LIN {X 0,Y 151.898,Z 448.046,A -85,B 0,C 180,E1 -25589.636,E2 -25589.636} C_VEL
LIN {X 0,Y 155.707,Z 455.378,A -85,B 0,C 180,E1 -25592.608,E2 -25592.608} C_VEL
LIN {X 0,Y 160.06,Z 464.974,A -85,B 0,C 180,E1 -25595.673,E2 -25595.673} C_VEL
LIN {X 0,Y 164.025,Z 475.268,A -85,B 0,C 180,E1 -25598.259,E2 -25598.259} C_VEL
LIN {X 0,Y 165.804,Z 480.611,A -85,B 0,C 180,E1 -25599.382,E2 -25599.382} C_VEL
LIN {X 0,Y 163.11,Z 515.862,A -85,B 0,C 180,E1 -25600.725,E2 -25600.725} C_VEL
LIN {X 0,Y 160.97,Z 529.245,A -85,B 0,C 180,E1 -25601.57,E2 -25601.57} C_VEL
LIN {X 0,Y 157.876,Z 541.895,A -85,B 0,C 180,E1 -25602.735,E2 -25602.735} C_VEL
LIN {X 0,Y 153.84,Z 554.553,A -85,B 0,C 180,E1 -25604.456,E2 -25604.456} C_VEL
LIN {X 0,Y 149.366,Z 565.815,A -85,B 0,C 180,E1 -25606.518,E2 -25606.518} C_VEL
LIN {X 0,Y 144.684,Z 575.966,A -85,B 0,C 180,E1 -25609.024,E2 -25609.024} C_VEL
LIN {X 0,Y 139.779,Z 585.115,A -85,B 0,C 180,E1 -25611.982,E2 -25611.982} C_VEL
LIN {X 0,Y 134.561,Z 594.043,A -85,B 0,C 180,E1 -25615.844,E2 -25615.844} C_VEL
LIN {X 0,Y 130.252,Z 601.039,A -85,B 0,C 180,E1 -25619.899,E2 -25619.899} C_VEL
LIN {X 0,Y 126.978,Z 606.098,A -85,B 0,C 180,E1 -25623.719,E2 -25623.719} C_VEL
LIN {X 0,Y 123.831,Z 610.825,A -85,B 0,C 180,E1 -25628.352,E2 -25628.352} C_VEL
LIN {X 0,Y 121.487,Z 614.442,A -85,B 0,C 180,E1 -25633.187,E2 -25633.187} C_VEL
LIN {X 0,Y 120.47,Z 616.313,A -85,B 0,C 180,E1 -25636.506,E2 -25636.506} C_VEL
LIN {X 0,Y 119.405,Z 618.728,A -85,B 0,C 180,E1 -25643.24,E2 -25643.24} C_VEL
LIN {X 0,Y 119.285,Z 619.346,A -85,B 0,C 180,E1 -25646.622,E2 -25646.622} C_VEL
LIN {X 0,Y 119.437,Z 619.565,A -85,B 0,C 180,E1 -25650,E2 -25650} C_VEL
LIN {X 0,Y 119.29,Z 619.33,A -85,B 0,C 180,E1 -25653.377,E2 -25653.377} C_VEL
LIN {X 0,Y 119.405,Z 618.702,A -85,B 0,C 180,E1 -25656.76,E2 -25656.76} C_VEL
LIN {X 0,Y 120.46,Z 616.26,A -85,B 0,C 180,E1 -25663.495,E2 -25663.495} C_VEL
LIN {X 0,Y 122.132,Z 613.287,A -85,B 0,C 180,E1 -25668.451,E2 -25668.451} C_VEL
LIN {X 0,Y 124.81,Z 609.284,A -85,B 0,C 180,E1 -25673.214,E2 -25673.214} C_VEL
LIN {X 0,Y 128.929,Z 603.138,A -85,B 0,C 180,E1 -25678.487,E2 -25678.487} C_VEL
LIN {X 0,Y 133.082,Z 596.427,A -85,B 0,C 180,E1 -25682.771,E2 -25682.771} C_VEL
LIN {X 0,Y 137.405,Z 589.092,A -85,B 0,C 180,E1 -25686.342,E2 -25686.342} C_VEL
LIN {X 0,Y 139.085,Z 585.217,A -85,B 0,C 180,E1 -25688.057,E2 -25688.057} C_VEL
LIN {X 0,Y 140.42,Z 578.568,A -85,B 0,C 180,E1 -25691.026,E2 -25691.026} C_VEL
LIN {X 0,Y 141.845,Z 571.485,A -85,B 0,C 180,E1 -25693.77,E2 -25693.77} C_VEL
LIN {X 0,Y 143.555,Z 566.815,A -85,B 0,C 180,E1 -25695.069,E2 -25695.069} C_VEL
LIN {X 0,Y 148.334,Z 555.407,A -85,B 0,C 180,E1 -25697.254,E2 -25697.254} C_VEL
LIN {X 0,Y 152.533,Z 543.035,A -85,B 0,C 180,E1 -25698.979,E2 -25698.979} C_VEL
LIN {X 0,Y 155.862,Z 530.29,A -85,B 0,C 180,E1 -25700.224,E2 -25700.224} C_VEL
LIN {X 0,Y 158.114,Z 517.266,A -85,B 0,C 180,E1 -25701.088,E2 -25701.088} C_VEL
LIN {X 0,Y 159.913,Z 497.723,A -85,B 0,C 180,E1 -25701.856,E2 -25701.856} C_VEL
LIN {X 0,Y 161.012,Z 482.58,A -85,B 0,C 180,E1 -25702.431,E2 -25702.431} C_VEL
LIN {X 0,Y 157.346,Z 472.01,A -85,B 0,C 180,E1 -25704.993,E2 -25704.993} C_VEL
LIN {X 0,Y 153.318,Z 462.421,A -85,B 0,C 180,E1 -25707.993,E2 -25707.993} C_VEL
LIN {X 0,Y 149.395,Z 454.26,A -85,B 0,C 180,E1 -25711.24,E2 -25711.24} C_VEL
LIN {X 0,Y 147.712,Z 451.268,A -85,B 0,C 180,E1 -25712.745,E2 -25712.745} C_VEL
LIN {X 0,Y 145.123,Z 447.379,A -85,B 0,C 180,E1 -25715.216,E2 -25715.216} C_VEL
LIN {X 0,Y 143.491,Z 445.063,A -85,B 0,C 180,E1 -25716.932,E2 -25716.932} C_VEL
LIN {X 0,Y 140.441,Z 440.755,A -85,B 0,C 180,E1 -25720.638,E2 -25720.638} C_VEL
LIN {X 0,Y 137.82,Z 437.299,A -85,B 0,C 180,E1 -25724.601,E2 -25724.601} C_VEL
LIN {X 0,Y 137.143,Z 435.979,A -85,B 0,C 180,E1 -25725.912,E2 -25725.912} C_VEL
LIN {X 0,Y 134.763,Z 433.642,A -85,B 0,C 180,E1 -25731.377,E2 -25731.377} C_VEL
LIN {X 0,Y 133.744,Z 430.501,A -85,B 0,C 180,E1 -25736.988,E2 -25736.988} C_VEL
LIN {X 0,Y 133.758,Z 430.581,A -85,B 0,C 180,E1 -25743.766,E2 -25743.766} C_VEL
LIN {X 0,Y 135.77,Z 435.019,A -85,B 0,C 180,E1 -25751.95,E2 -25751.95} C_VEL
LIN {X 0,Y 137.421,Z 436.418,A -85,B 0,C 180,E1 -25755.195,E2 -25755.195} C_VEL
LIN {X 0,Y 139.584,Z 439.959,A -85,B 0,C 180,E1 -25758.801,E2 -25758.801} C_VEL
LIN {X 0,Y 141.075,Z 441.564,A -85,B 0,C 180,E1 -25760.762,E2 -25760.762} C_VEL
LIN {X 0,Y 143.801,Z 445.413,A -85,B 0,C 180,E1 -25763.97,E2 -25763.97} C_VEL
LIN {X 0,Y 147.607,Z 451.079,A -85,B 0,C 180,E1 -25767.731,E2 -25767.731} C_VEL
LIN {X 0,Y 151.619,Z 457.249,A -85,B 0,C 180,E1 -25771.085,E2 -25771.085} C_VEL
LIN {X 0,Y 156.549,Z 466.058,A -85,B 0,C 180,E1 -25774.697,E2 -25774.697} C_VEL
LIN {X 0,Y 161.36,Z 475.703,A -85,B 0,C 180,E1 -25777.813,E2 -25777.813} C_VEL
LIN {X 0,Y 161.39,Z 478.372,A -85,B 0,C 180,E1 -25778.017,E2 -25778.017} C_VEL
LIN {X 0,Y 158.8,Z 508.594,A -85,B 0,C 180,E1 -25779.135,E2 -25779.135} C_VEL
LIN {X 0,Y 156.693,Z 521.604,A -85,B 0,C 180,E1 -25779.997,E2 -25779.997} C_VEL
LIN {X 0,Y 153.789,Z 534.273,A -85,B 0,C 180,E1 -25781.309,E2 -25781.309} C_VEL
LIN {X 0,Y 150.119,Z 546.042,A -85,B 0,C 180,E1 -25782.989,E2 -25782.989} C_VEL
LIN {X 0,Y 145.681,Z 557.357,A -85,B 0,C 180,E1 -25785.128,E2 -25785.128} C_VEL
LIN {X 0,Y 140.907,Z 567.552,A -85,B 0,C 180,E1 -25787.676,E2 -25787.676} C_VEL
LIN {X 0,Y 135.995,Z 576.857,A -85,B 0,C 180,E1 -25790.821,E2 -25790.821} C_VEL
LIN {X 0,Y 130.749,Z 585.578,A -85,B 0,C 180,E1 -25794.703,E2 -25794.703} C_VEL
LIN {X 0,Y 125.877,Z 592.732,A -85,B 0,C 180,E1 -25798.906,E2 -25798.906} C_VEL
LIN {X 0,Y 122.303,Z 597.552,A -85,B 0,C 180,E1 -25802.632,E2 -25802.632} C_VEL
LIN {X 0,Y 118.814,Z 602.229,A -85,B 0,C 180,E1 -25807.389,E2 -25807.389} C_VEL
LIN {X 0,Y 116.072,Z 605.804,A -85,B 0,C 180,E1 -25812.378,E2 -25812.378} C_VEL
LIN {X 0,Y 114.68,Z 607.648,A -85,B 0,C 180,E1 -25815.811,E2 -25815.811} C_VEL
LIN {X 0,Y 113.655,Z 609.03,A -85,B 0,C 180,E1 -25819.309,E2 -25819.309} C_VEL
LIN {X 0,Y 112.554,Z 610.615,A -85,B 0,C 180,E1 -25826.42,E2 -25826.42} C_VEL
LIN {X 0,Y 112.46,Z 610.815,A -85,B 0,C 180,E1 -25830.805,E2 -25830.805} C_VEL
LIN {X 0,Y 112.937,Z 610.06,A -85,B 0,C 180,E1 -25837.149,E2 -25837.149} C_VEL
LIN {X 0,Y 113.655,Z 609.095,A -85,B 0,C 180,E1 -25840.691,E2 -25840.691} C_VEL
LIN {X 0,Y 114.681,Z 607.741,A -85,B 0,C 180,E1 -25844.189,E2 -25844.189} C_VEL
LIN {X 0,Y 116.889,Z 604.878,A -85,B 0,C 180,E1 -25849.31,E2 -25849.31} C_VEL
LIN {X 0,Y 119.884,Z 600.992,A -85,B 0,C 180,E1 -25854.227,E2 -25854.227} C_VEL
LIN {X 0,Y 123.62,Z 595.977,A -85,B 0,C 180,E1 -25858.896,E2 -25858.896} C_VEL
LIN {X 0,Y 128.157,Z 589.65,A -85,B 0,C 180,E1 -25863.256,E2 -25863.256} C_VEL
LIN {X 0,Y 132.997,Z 582.238,A -85,B 0,C 180,E1 -25867.098,E2 -25867.098} C_VEL
LIN {X 0,Y 137.732,Z 573.85,A -85,B 0,C 180,E1 -25870.489,E2 -25870.489} C_VEL
LIN {X 0,Y 142.858,Z 563.823,A -85,B 0,C 180,E1 -25873.529,E2 -25873.529} C_VEL
LIN {X 0,Y 147.78,Z 552.715,A -85,B 0,C 180,E1 -25875.996,E2 -25875.996} C_VEL
LIN {X 0,Y 151.746,Z 541.824,A -85,B 0,C 180,E1 -25877.818,E2 -25877.818} C_VEL
LIN {X 0,Y 155.166,Z 529.783,A -85,B 0,C 180,E1 -25879.345,E2 -25879.345} C_VEL
LIN {X 0,Y 157.745,Z 517.548,A -85,B 0,C 180,E1 -25880.442,E2 -25880.442} C_VEL
LIN {X 0,Y 159.469,Z 504.548,A -85,B 0,C 180,E1 -25881.198,E2 -25881.198} C_VEL
LIN {X 0,Y 161.719,Z 476.236,A -85,B 0,C 180,E1 -25882.227,E2 -25882.227} C_VEL
LIN {X 0,Y 156.559,Z 465.823,A -85,B 0,C 180,E1 -25885.583,E2 -25885.583} C_VEL
LIN {X 0,Y 151.591,Z 457.083,A -85,B 0,C 180,E1 -25889.245,E2 -25889.245} C_VEL
LIN {X 0,Y 146.672,Z 449.456,A -85,B 0,C 180,E1 -25893.498,E2 -25893.498} C_VEL
LIN {X 0,Y 143.599,Z 445.106,A -85,B 0,C 180,E1 -25896.642,E2 -25896.642} C_VEL
LIN {X 0,Y 140.633,Z 440.871,A -85,B 0,C 180,E1 -25900.286,E2 -25900.286} C_VEL
LIN {X 0,Y 138.148,Z 437.792,A -85,B 0,C 180,E1 -25904.017,E2 -25904.017} C_VEL
LIN {X 0,Y 137.268,Z 436.076,A -85,B 0,C 180,E1 -25905.735,E2 -25905.735} C_VEL
LIN {X 0,Y 134.495,Z 432.997,A -85,B 0,C 180,E1 -25912.984,E2 -25912.984} C_VEL
LIN {X 0,Y 133.934,Z 430.588,A -85,B 0,C 180,E1 -25917.744,E2 -25917.744} C_VEL
LIN {X 0,Y 133.942,Z 430.596,A -85,B 0,C 180,E1 -25921.879,E2 -25921.879} C_VEL
LIN {X 0,Y 135.847,Z 434.983,A -85,B 0,C 180,E1 -25930.844,E2 -25930.844} C_VEL
LIN {X 0,Y 137.55,Z 436.503,A -85,B 0,C 180,E1 -25934.329,E2 -25934.329} C_VEL
LIN {X 0,Y 139.682,Z 439.963,A -85,B 0,C 180,E1 -25937.949,E2 -25937.949} C_VEL
LIN {X 0,Y 141.148,Z 441.629,A -85,B 0,C 180,E1 -25939.923,E2 -25939.923} C_VEL
LIN {X 0,Y 143.897,Z 445.421,A -85,B 0,C 180,E1 -25943.19,E2 -25943.19} C_VEL
LIN {X 0,Y 147.428,Z 450.703,A -85,B 0,C 180,E1 -25946.739,E2 -25946.739} C_VEL
LIN {X 0,Y 149.328,Z 453.968,A -85,B 0,C 180,E1 -25948.459,E2 -25948.459} C_VEL
LIN {X 0,Y 152.788,Z 461.003,A -85,B 0,C 180,E1 -25951.369,E2 -25951.369} C_VEL
LIN {X 0,Y 156.686,Z 470.102,A -85,B 0,C 180,E1 -25954.341,E2 -25954.341} C_VEL
LIN {X 0,Y 160.073,Z 479.33,A -85,B 0,C 180,E1 -25956.742,E2 -25956.742} C_VEL
LIN {X 0,Y 161.203,Z 482.769,A -85,B 0,C 180,E1 -25957.517,E2 -25957.517} C_VEL
LIN {X 0,Y 158.541,Z 515.781,A -85,B 0,C 180,E1 -25958.787,E2 -25958.787} C_VEL
LIN {X 0,Y 156.281,Z 529.32,A -85,B 0,C 180,E1 -25959.648,E2 -25959.648} C_VEL
LIN {X 0,Y 153.15,Z 541.635,A -85,B 0,C 180,E1 -25960.785,E2 -25960.785} C_VEL
LIN {X 0,Y 148.957,Z 554.291,A -85,B 0,C 180,E1 -25962.507,E2 -25962.507} C_VEL
LIN {X 0,Y 144.286,Z 565.552,A -85,B 0,C 180,E1 -25964.573,E2 -25964.573} C_VEL
LIN {X 0,Y 139.393,Z 575.701,A -85,B 0,C 180,E1 -25967.107,E2 -25967.107} C_VEL
LIN {X 0,Y 134.236,Z 584.849,A -85,B 0,C 180,E1 -25970.108,E2 -25970.108} C_VEL
LIN {X 0,Y 128.719,Z 593.777,A -85,B 0,C 180,E1 -25974.061,E2 -25974.061} C_VEL
LIN {X 0,Y 124.382,Z 600.333,A -85,B 0,C 180,E1 -25977.946,E2 -25977.946} C_VEL
LIN {X 0,Y 120.638,Z 605.831,A -85,B 0,C 180,E1 -25982.222,E2 -25982.222} C_VEL
LIN {X 0,Y 117.223,Z 610.557,A -85,B 0,C 180,E1 -25987.065,E2 -25987.065} C_VEL
LIN {X 0,Y 114.657,Z 614.174,A -85,B 0,C 180,E1 -25992.153,E2 -25992.153} C_VEL
LIN {X 0,Y 113.542,Z 616.045,A -85,B 0,C 180,E1 -25995.665,E2 -25995.665} C_VEL
LIN {X 0,Y 112.326,Z 618.46,A -85,B 0,C 180,E1 -26002.812,E2 -26002.812} C_VEL
LIN {X 0,Y 112.202,Z 619.079,A -85,B 0,C 180,E1 -26006.409,E2 -26006.409} C_VEL
LIN {X 0,Y 112.338,Z 619.298,A -85,B 0,C 180,E1 -26010,E2 -26010} C_VEL
LIN {X 0,Y 112.205,Z 619.062,A -85,B 0,C 180,E1 -26013.591,E2 -26013.591} C_VEL
LIN {X 0,Y 112.325,Z 618.434,A -85,B 0,C 180,E1 -26017.188,E2 -26017.188} C_VEL
LIN {X 0,Y 112.737,Z 617.414,A -85,B 0,C 180,E1 -26020.779,E2 -26020.779} C_VEL
LIN {X 0,Y 113.534,Z 615.991,A -85,B 0,C 180,E1 -26024.336,E2 -26024.336} C_VEL
LIN {X 0,Y 115.392,Z 613.018,A -85,B 0,C 180,E1 -26029.571,E2 -26029.571} C_VEL
LIN {X 0,Y 118.299,Z 609.015,A -85,B 0,C 180,E1 -26034.573,E2 -26034.573} C_VEL
LIN {X 0,Y 122.704,Z 602.868,A -85,B 0,C 180,E1 -26040.076,E2 -26040.076} C_VEL
LIN {X 0,Y 127.137,Z 596.157,A -85,B 0,C 180,E1 -26044.513,E2 -26044.513} C_VEL
LIN {X 0,Y 132.349,Z 587.844,A -85,B 0,C 180,E1 -26048.604,E2 -26048.604} C_VEL
LIN {X 0,Y 137.296,Z 579.326,A -85,B 0,C 180,E1 -26051.716,E2 -26051.716} C_VEL
LIN {X 0,Y 142.618,Z 568.805,A -85,B 0,C 180,E1 -26054.604,E2 -26054.604} C_VEL
LIN {X 0,Y 143.555,Z 566.815,A -85,B 0,C 180,E1 -26055.069,E2 -26055.069} C_VEL
LIN {X 0,Y 145.242,Z 562.044,A -85,B 0,C 180,E1 -26056.287,E2 -26056.287} C_VEL
LIN {X 0,Y 146.535,Z 554.03,A -85,B 0,C 180,E1 -26058.535,E2 -26058.535} C_VEL
LIN {X 0,Y 147.564,Z 545.615,A -85,B 0,C 180,E1 -26060.534,E2 -26060.534} C_VEL
LIN {X 0,Y 148.757,Z 540.218,A -85,B 0,C 180,E1 -26061.335,E2 -26061.335} C_VEL
LIN {X 0,Y 152.106,Z 526.668,A -85,B 0,C 180,E1 -26062.548,E2 -26062.548} C_VEL
LIN {X 0,Y 154.184,Z 513.808,A -85,B 0,C 180,E1 -26063.306,E2 -26063.306} C_VEL
LIN {X 0,Y 156.57,Z 484.854,A -85,B 0,C 180,E1 -26064.399,E2 -26064.399} C_VEL
LIN {X 0,Y 153.21,Z 474.95,A -85,B 0,C 180,E1 -26066.994,E2 -26066.994} C_VEL
LIN {X 0,Y 149.377,Z 465.489,A -85,B 0,C 180,E1 -26070.181,E2 -26070.181} C_VEL
LIN {X 0,Y 145.904,Z 458.145,A -85,B 0,C 180,E1 -26073.396,E2 -26073.396} C_VEL
LIN {X 0,Y 143.436,Z 454.246,A -85,B 0,C 180,E1 -26075.869,E2 -26075.869} C_VEL
LIN {X 0,Y 141.433,Z 451.219,A -85,B 0,C 180,E1 -26078.119,E2 -26078.119} C_VEL
LIN {X 0,Y 138.81,Z 447.332,A -85,B 0,C 180,E1 -26081.552,E2 -26081.552} C_VEL
LIN {X 0,Y 136.369,Z 443.881,A -85,B 0,C 180,E1 -26085.544,E2 -26085.544} C_VEL
LIN {X 0,Y 135.894,Z 442.878,A -85,B 0,C 180,E1 -26086.542,E2 -26086.542} C_VEL
LIN {X 0,Y 133.479,Z 440.082,A -85,B 0,C 180,E1 -26092.816,E2 -26092.816} C_VEL
LIN {X 0,Y 132.794,Z 437.51,A -85,B 0,C 180,E1 -26097.725,E2 -26097.725} C_VEL
LIN {X 0,Y 132.81,Z 437.541,A -85,B 0,C 180,E1 -26103.034,E2 -26103.034} C_VEL
LIN {X 0,Y 134.912,Z 442.167,A -85,B 0,C 180,E1 -26112.027,E2 -26112.027} C_VEL
LIN {X 0,Y 136.068,Z 443.179,A -85,B 0,C 180,E1 -26114.393,E2 -26114.393} C_VEL
LIN {X 0,Y 138.336,Z 446.887,A -85,B 0,C 180,E1 -26118.361,E2 -26118.361} C_VEL
LIN {X 0,Y 139.495,Z 448.297,A -85,B 0,C 180,E1 -26119.979,E2 -26119.979} C_VEL
LIN {X 0,Y 142.676,Z 453.086,A -85,B 0,C 180,E1 -26123.882,E2 -26123.882} C_VEL
LIN {X 0,Y 145.471,Z 457.457,A -85,B 0,C 180,E1 -26126.765,E2 -26126.765} C_VEL
LIN {X 0,Y 149.169,Z 463.467,A -85,B 0,C 180,E1 -26130.064,E2 -26130.064} C_VEL
LIN {X 0,Y 153.361,Z 471.307,A -85,B 0,C 180,E1 -26133.362,E2 -26133.362} C_VEL
LIN {X 0,Y 157.046,Z 478.923,A -85,B 0,C 180,E1 -26135.961,E2 -26135.961} C_VEL
LIN {X 0,Y 154.445,Z 508.748,A -85,B 0,C 180,E1 -26137.089,E2 -26137.089} C_VEL
LIN {X 0,Y 152.179,Z 522.161,A -85,B 0,C 180,E1 -26137.976,E2 -26137.976} C_VEL
LIN {X 0,Y 149.214,Z 534.546,A -85,B 0,C 180,E1 -26139.268,E2 -26139.268} C_VEL
LIN {X 0,Y 145.374,Z 546.314,A -85,B 0,C 180,E1 -26140.943,E2 -26140.943} C_VEL
LIN {X 0,Y 140.752,Z 557.628,A -85,B 0,C 180,E1 -26143.094,E2 -26143.094} C_VEL
LIN {X 0,Y 135.762,Z 567.821,A -85,B 0,C 180,E1 -26145.666,E2 -26145.666} C_VEL
LIN {X 0,Y 130.221,Z 577.69,A -85,B 0,C 180,E1 -26149.076,E2 -26149.076} C_VEL
LIN {X 0,Y 125.03,Z 585.847,A -85,B 0,C 180,E1 -26152.825,E2 -26152.825} C_VEL
LIN {X 0,Y 119.869,Z 593,A -85,B 0,C 180,E1 -26157.158,E2 -26157.158} C_VEL
LIN {X 0,Y 116.038,Z 597.821,A -85,B 0,C 180,E1 -26161.019,E2 -26161.019} C_VEL
LIN {X 0,Y 112.296,Z 602.497,A -85,B 0,C 180,E1 -26165.997,E2 -26165.997} C_VEL
LIN {X 0,Y 109.343,Z 606.071,A -85,B 0,C 180,E1 -26171.254,E2 -26171.254} C_VEL
LIN {X 0,Y 107.806,Z 607.916,A -85,B 0,C 180,E1 -26174.885,E2 -26174.885} C_VEL
LIN {X 0,Y 106.682,Z 609.298,A -85,B 0,C 180,E1 -26178.602,E2 -26178.602} C_VEL
LIN {X 0,Y 105.921,Z 610.28,A -85,B 0,C 180,E1 -26182.374,E2 -26182.374} C_VEL
LIN {X 0,Y 105.392,Z 611.105,A -85,B 0,C 180,E1 -26190,E2 -26190} C_VEL
LIN {X 0,Y 105.47,Z 610.911,A -85,B 0,C 180,E1 -26193.821,E2 -26193.821} C_VEL
LIN {X 0,Y 105.921,Z 610.326,A -85,B 0,C 180,E1 -26197.626,E2 -26197.626} C_VEL
LIN {X 0,Y 107.805,Z 608.008,A -85,B 0,C 180,E1 -26205.115,E2 -26205.115} C_VEL
LIN {X 0,Y 110.209,Z 605.145,A -85,B 0,C 180,E1 -26210.532,E2 -26210.532} C_VEL
LIN {X 0,Y 113.438,Z 601.258,A -85,B 0,C 180,E1 -26215.701,E2 -26215.701} C_VEL
LIN {X 0,Y 117.443,Z 596.243,A -85,B 0,C 180,E1 -26220.574,E2 -26220.574} C_VEL
LIN {X 0,Y 122.3,Z 589.914,A -85,B 0,C 180,E1 -26225.074,E2 -26225.074} C_VEL
LIN {X 0,Y 127.236,Z 582.763,A -85,B 0,C 180,E1 -26228.907,E2 -26228.907} C_VEL
LIN {X 0,Y 132.514,Z 573.937,A -85,B 0,C 180,E1 -26232.547,E2 -26232.547} C_VEL
LIN {X 0,Y 137.813,Z 564.086,A -85,B 0,C 180,E1 -26235.556,E2 -26235.556} C_VEL
LIN {X 0,Y 142.946,Z 552.977,A -85,B 0,C 180,E1 -26238.04,E2 -26238.04} C_VEL
LIN {X 0,Y 147.082,Z 542.085,A -85,B 0,C 180,E1 -26239.863,E2 -26239.863} C_VEL
LIN {X 0,Y 150.649,Z 530.042,A -85,B 0,C 180,E1 -26241.389,E2 -26241.389} C_VEL
LIN {X 0,Y 153.297,Z 517.953,A -85,B 0,C 180,E1 -26242.476,E2 -26242.476} C_VEL
LIN {X 0,Y 155.125,Z 504.764,A -85,B 0,C 180,E1 -26243.242,E2 -26243.242} C_VEL
LIN {X 0,Y 157.251,Z 479.098,A -85,B 0,C 180,E1 -26244.18,E2 -26244.18} C_VEL
LIN {X 0,Y 152.39,Z 469.167,A -85,B 0,C 180,E1 -26247.674,E2 -26247.674} C_VEL
LIN {X 0,Y 148.283,Z 461.816,A -85,B 0,C 180,E1 -26251.019,E2 -26251.019} C_VEL
LIN {X 0,Y 144.468,Z 455.612,A -85,B 0,C 180,E1 -26254.614,E2 -26254.614} C_VEL
LIN {X 0,Y 141.872,Z 451.708,A -85,B 0,C 180,E1 -26257.455,E2 -26257.455} C_VEL
LIN {X 0,Y 139.007,Z 447.486,A -85,B 0,C 180,E1 -26261.197,E2 -26261.197} C_VEL
LIN {X 0,Y 136.536,Z 444.053,A -85,B 0,C 180,E1 -26265.277,E2 -26265.277} C_VEL
LIN {X 0,Y 135.939,Z 442.892,A -85,B 0,C 180,E1 -26266.547,E2 -26266.547} C_VEL
LIN {X 0,Y 133.113,Z 438.671,A -85,B 0,C 180,E1 -26276.216,E2 -26276.216} C_VEL
LIN {X 0,Y 133.03,Z 437.547,A -85,B 0,C 180,E1 -26278.486,E2 -26278.486} C_VEL
LIN {X 0,Y 133.044,Z 437.791,A -85,B 0,C 180,E1 -26281.703,E2 -26281.703} C_VEL
LIN {X 0,Y 135.454,Z 442.537,A -85,B 0,C 180,E1 -26291.978,E2 -26291.978} C_VEL
LIN {X 0,Y 136.251,Z 443.328,A -85,B 0,C 180,E1 -26293.612,E2 -26293.612} C_VEL
LIN {X 0,Y 138.325,Z 446.772,A -85,B 0,C 180,E1 -26297.338,E2 -26297.338} C_VEL
LIN {X 0,Y 139.495,Z 448.226,A -85,B 0,C 180,E1 -26299.02,E2 -26299.02} C_VEL
LIN {X 0,Y 142.623,Z 452.852,A -85,B 0,C 180,E1 -26302.929,E2 -26302.929} C_VEL
LIN {X 0,Y 145.427,Z 457.261,A -85,B 0,C 180,E1 -26305.876,E2 -26305.876} C_VEL
LIN {X 0,Y 147.435,Z 461.072,A -85,B 0,C 180,E1 -26307.814,E2 -26307.814} C_VEL
LIN {X 0,Y 151.011,Z 469.051,A -85,B 0,C 180,E1 -26310.987,E2 -26310.987} C_VEL
LIN {X 0,Y 154.599,Z 478.492,A -85,B 0,C 180,E1 -26313.889,E2 -26313.889} C_VEL
LIN {X 0,Y 156.772,Z 485.135,A -85,B 0,C 180,E1 -26315.556,E2 -26315.556} C_VEL
LIN {X 0,Y 154.16,Z 515.837,A -85,B 0,C 180,E1 -26316.751,E2 -26316.751} C_VEL
LIN {X 0,Y 151.775,Z 529.42,A -85,B 0,C 180,E1 -26317.612,E2 -26317.612} C_VEL
LIN {X 0,Y 148.613,Z 541.374,A -85,B 0,C 180,E1 -26318.714,E2 -26318.714} C_VEL
LIN {X 0,Y 144.255,Z 554.028,A -85,B 0,C 180,E1 -26320.428,E2 -26320.428} C_VEL
LIN {X 0,Y 139.375,Z 565.287,A -85,B 0,C 180,E1 -26322.485,E2 -26322.485} C_VEL
LIN {X 0,Y 134.265,Z 575.436,A -85,B 0,C 180,E1 -26325.039,E2 -26325.039} C_VEL
LIN {X 0,Y 128.86,Z 584.584,A -85,B 0,C 180,E1 -26328.08,E2 -26328.08} C_VEL
LIN {X 0,Y 123.008,Z 593.51,A -85,B 0,C 180,E1 -26332.108,E2 -26332.108} C_VEL
LIN {X 0,Y 117.969,Z 600.655,A -85,B 0,C 180,E1 -26336.517,E2 -26336.517} C_VEL
LIN {X 0,Y 114.394,Z 605.565,A -85,B 0,C 180,E1 -26340.562,E2 -26340.562} C_VEL
LIN {X 0,Y 110.689,Z 610.29,A -85,B 0,C 180,E1 -26345.626,E2 -26345.626} C_VEL
LIN {X 0,Y 107.876,Z 613.905,A -85,B 0,C 180,E1 -26350.99,E2 -26350.99} C_VEL
LIN {X 0,Y 106.627,Z 615.777,A -85,B 0,C 180,E1 -26354.714,E2 -26354.714} C_VEL
LIN {X 0,Y 105.764,Z 617.184,A -85,B 0,C 180,E1 -26358.501,E2 -26358.501} C_VEL
LIN {X 0,Y 105.268,Z 618.193,A -85,B 0,C 180,E1 -26362.327,E2 -26362.327} C_VEL
LIN {X 0,Y 105.11,Z 618.812,A -85,B 0,C 180,E1 -26366.166,E2 -26366.166} C_VEL
LIN {X 0,Y 105.235,Z 619.031,A -85,B 0,C 180,E1 -26370,E2 -26370} C_VEL
LIN {X 0,Y 105.112,Z 618.795,A -85,B 0,C 180,E1 -26373.834,E2 -26373.834} C_VEL
LIN {X 0,Y 105.266,Z 618.165,A -85,B 0,C 180,E1 -26377.673,E2 -26377.673} C_VEL
LIN {X 0,Y 105.759,Z 617.146,A -85,B 0,C 180,E1 -26381.499,E2 -26381.499} C_VEL
LIN {X 0,Y 106.62,Z 615.721,A -85,B 0,C 180,E1 -26385.287,E2 -26385.287} C_VEL
LIN {X 0,Y 108.71,Z 612.749,A -85,B 0,C 180,E1 -26390.828,E2 -26390.828} C_VEL
LIN {X 0,Y 111.844,Z 608.745,A -85,B 0,C 180,E1 -26396.095,E2 -26396.095} C_VEL
LIN {X 0,Y 116.577,Z 602.597,A -85,B 0,C 180,E1 -26401.836,E2 -26401.836} C_VEL
LIN {X 0,Y 121.317,Z 595.886,A -85,B 0,C 180,E1 -26406.426,E2 -26406.426} C_VEL
LIN {X 0,Y 126.874,Z 587.574,A -85,B 0,C 180,E1 -26410.606,E2 -26410.606} C_VEL
LIN {X 0,Y 132.069,Z 579.055,A -85,B 0,C 180,E1 -26413.771,E2 -26413.771} C_VEL
LIN {X 0,Y 137.654,Z 568.535,A -85,B 0,C 180,E1 -26416.679,E2 -26416.679} C_VEL
LIN {X 0,Y 142.984,Z 556.693,A -85,B 0,C 180,E1 -26419.086,E2 -26419.086} C_VEL
LIN {X 0,Y 147.346,Z 544.754,A -85,B 0,C 180,E1 -26420.81,E2 -26420.81} C_VEL
LIN {X 0,Y 148.757,Z 540.218,A -85,B 0,C 180,E1 -26421.335,E2 -26421.335} C_VEL
LIN {X 0,Y 149.88,Z 534.719,A -85,B 0,C 180,E1 -26422.069,E2 -26422.069} C_VEL
LIN {X 0,Y 150.027,Z 522.125,A -85,B 0,C 180,E1 -26424.338,E2 -26424.338} C_VEL
LIN {X 0,Y 150.061,Z 514.66,A -85,B 0,C 180,E1 -26425.337,E2 -26425.337} C_VEL
LIN {X 0,Y 150.36,Z 510.79,A -85,B 0,C 180,E1 -26425.58,E2 -26425.58} C_VEL
LIN {X 0,Y 152.323,Z 487.133,A -85,B 0,C 180,E1 -26426.48,E2 -26426.48} C_VEL
LIN {X 0,Y 149.348,Z 478.239,A -85,B 0,C 180,E1 -26429.023,E2 -26429.023} C_VEL
LIN {X 0,Y 146.351,Z 470.432,A -85,B 0,C 180,E1 -26431.79,E2 -26431.79} C_VEL
LIN {X 0,Y 143.309,Z 463.671,A -85,B 0,C 180,E1 -26434.88,E2 -26434.88} C_VEL
LIN {X 0,Y 139.989,Z 458.128,A -85,B 0,C 180,E1 -26438.655,E2 -26438.655} C_VEL
LIN {X 0,Y 137.095,Z 453.802,A -85,B 0,C 180,E1 -26442.664,E2 -26442.664} C_VEL
LIN {X 0,Y 134.762,Z 449.983,A -85,B 0,C 180,E1 -26446.955,E2 -26446.955} C_VEL
LIN {X 0,Y 131.932,Z 444.884,A -85,B 0,C 180,E1 -26457.329,E2 -26457.329} C_VEL
LIN {X 0,Y 131.814,Z 444.427,A -85,B 0,C 180,E1 -26460,E2 -26460} C_VEL
LIN {X 0,Y 131.923,Z 444.776,A -85,B 0,C 180,E1 -26463.054,E2 -26463.054} C_VEL
LIN {X 0,Y 134.056,Z 449.297,A -85,B 0,C 180,E1 -26472.105,E2 -26472.105} C_VEL
LIN {X 0,Y 134.82,Z 450.138,A -85,B 0,C 180,E1 -26473.759,E2 -26473.759} C_VEL
LIN {X 0,Y 137.286,Z 454.029,A -85,B 0,C 180,E1 -26478.197,E2 -26478.197} C_VEL
LIN {X 0,Y 140.755,Z 459.431,A -85,B 0,C 180,E1 -26482.863,E2 -26482.863} C_VEL
LIN {X 0,Y 144.514,Z 465.551,A -85,B 0,C 180,E1 -26486.887,E2 -26486.887} C_VEL
LIN {X 0,Y 148.938,Z 473.731,A -85,B 0,C 180,E1 -26490.875,E2 -26490.875} C_VEL
LIN {X 0,Y 152.737,Z 481.739,A -85,B 0,C 180,E1 -26493.879,E2 -26493.879} C_VEL
LIN {X 0,Y 150.318,Z 508.789,A -85,B 0,C 180,E1 -26494.925,E2 -26494.925} C_VEL
LIN {X 0,Y 148.008,Z 522.046,A -85,B 0,C 180,E1 -26495.782,E2 -26495.782} C_VEL
LIN {X 0,Y 144.841,Z 534.819,A -85,B 0,C 180,E1 -26497.102,E2 -26497.102} C_VEL
LIN {X 0,Y 140.832,Z 546.586,A -85,B 0,C 180,E1 -26498.765,E2 -26498.765} C_VEL
LIN {X 0,Y 136.016,Z 557.898,A -85,B 0,C 180,E1 -26500.917,E2 -26500.917} C_VEL
LIN {X 0,Y 130.79,Z 568.091,A -85,B 0,C 180,E1 -26503.497,E2 -26503.497} C_VEL
LIN {X 0,Y 125.32,Z 577.396,A -85,B 0,C 180,E1 -26506.721,E2 -26506.721} C_VEL
LIN {X 0,Y 119.445,Z 586.117,A -85,B 0,C 180,E1 -26510.765,E2 -26510.765} C_VEL
LIN {X 0,Y 113.987,Z 593.268,A -85,B 0,C 180,E1 -26515.229,E2 -26515.229} C_VEL
LIN {X 0,Y 109.877,Z 598.09,A -85,B 0,C 180,E1 -26519.224,E2 -26519.224} C_VEL
LIN {X 0,Y 105.855,Z 602.765,A -85,B 0,C 180,E1 -26524.434,E2 -26524.434} C_VEL
LIN {X 0,Y 102.635,Z 606.34,A -85,B 0,C 180,E1 -26529.979,E2 -26529.979} C_VEL
LIN {X 0,Y 100.976,Z 608.183,A -85,B 0,C 180,E1 -26533.836,E2 -26533.836} C_VEL
LIN {X 0,Y 99.745,Z 609.565,A -85,B 0,C 180,E1 -26537.797,E2 -26537.797} C_VEL
LIN {X 0,Y 98.4,Z 611.149,A -85,B 0,C 180,E1 -26545.904,E2 -26545.904} C_VEL
LIN {X 0,Y 98.311,Z 611.371,A -85,B 0,C 180,E1 -26550,E2 -26550} C_VEL
LIN {X 0,Y 98.4,Z 611.177,A -85,B 0,C 180,E1 -26554.096,E2 -26554.096} C_VEL
LIN {X 0,Y 99.745,Z 609.628,A -85,B 0,C 180,E1 -26562.203,E2 -26562.203} C_VEL
LIN {X 0,Y 100.973,Z 608.274,A -85,B 0,C 180,E1 -26566.165,E2 -26566.165} C_VEL
LIN {X 0,Y 103.578,Z 605.412,A -85,B 0,C 180,E1 -26571.912,E2 -26571.912} C_VEL
LIN {X 0,Y 107.081,Z 601.525,A -85,B 0,C 180,E1 -26577.35,E2 -26577.35} C_VEL
LIN {X 0,Y 111.38,Z 596.509,A -85,B 0,C 180,E1 -26582.434,E2 -26582.434} C_VEL
LIN {X 0,Y 116.564,Z 590.179,A -85,B 0,C 180,E1 -26587.079,E2 -26587.079} C_VEL
LIN {X 0,Y 121.468,Z 583.518,A -85,B 0,C 180,E1 -26590.775,E2 -26590.775} C_VEL
LIN {X 0,Y 126.301,Z 575.974,A -85,B 0,C 180,E1 -26594.07,E2 -26594.07} C_VEL
LIN {X 0,Y 132.374,Z 565.414,A -85,B 0,C 180,E1 -26597.445,E2 -26597.445} C_VEL
LIN {X 0,Y 137.724,Z 554.637,A -85,B 0,C 180,E1 -26599.945,E2 -26599.945} C_VEL
LIN {X 0,Y 142.019,Z 544.105,A -85,B 0,C 180,E1 -26601.774,E2 -26601.774} C_VEL
LIN {X 0,Y 146.031,Z 531.427,A -85,B 0,C 180,E1 -26603.427,E2 -26603.427} C_VEL
LIN {X 0,Y 148.971,Z 518.751,A -85,B 0,C 180,E1 -26604.603,E2 -26604.603} C_VEL
LIN {X 0,Y 150.911,Z 505.919,A -85,B 0,C 180,E1 -26605.352,E2 -26605.352} C_VEL
LIN {X 0,Y 152.953,Z 482.001,A -85,B 0,C 180,E1 -26606.254,E2 -26606.254} C_VEL
LIN {X 0,Y 148.809,Z 473.292,A -85,B 0,C 180,E1 -26609.555,E2 -26609.555} C_VEL
LIN {X 0,Y 145.267,Z 466.78,A -85,B 0,C 180,E1 -26612.735,E2 -26612.735} C_VEL
LIN {X 0,Y 141.901,Z 461.115,A -85,B 0,C 180,E1 -26616.23,E2 -26616.23} C_VEL
LIN {X 0,Y 139.806,Z 457.848,A -85,B 0,C 180,E1 -26618.74,E2 -26618.74} C_VEL
LIN {X 0,Y 137.306,Z 453.957,A -85,B 0,C 180,E1 -26622.301,E2 -26622.301} C_VEL
LIN {X 0,Y 135.044,Z 450.387,A -85,B 0,C 180,E1 -26626.456,E2 -26626.456} C_VEL
LIN {X 0,Y 134.55,Z 449.655,A -85,B 0,C 180,E1 -26627.557,E2 -26627.557} C_VEL
LIN {X 0,Y 132.153,Z 444.774,A -85,B 0,C 180,E1 -26638.294,E2 -26638.294} C_VEL
LIN {X 0,Y 132.146,Z 444.606,A -85,B 0,C 180,E1 -26640.626,E2 -26640.626} C_VEL
LIN {X 0,Y 134.597,Z 449.673,A -85,B 0,C 180,E1 -26652.056,E2 -26652.056} C_VEL
LIN {X 0,Y 135.111,Z 450.485,A -85,B 0,C 180,E1 -26653.202,E2 -26653.202} C_VEL
LIN {X 0,Y 137.101,Z 453.699,A -85,B 0,C 180,E1 -26656.896,E2 -26656.896} C_VEL
LIN {X 0,Y 137.936,Z 454.923,A -85,B 0,C 180,E1 -26658.184,E2 -26658.184} C_VEL
LIN {X 0,Y 140.854,Z 459.462,A -85,B 0,C 180,E1 -26662.072,E2 -26662.072} C_VEL
LIN {X 0,Y 143.546,Z 463.923,A -85,B 0,C 180,E1 -26665.075,E2 -26665.075} C_VEL
LIN {X 0,Y 146.594,Z 470.684,A -85,B 0,C 180,E1 -26668.176,E2 -26668.176} C_VEL
LIN {X 0,Y 149.921,Z 479.421,A -85,B 0,C 180,E1 -26671.238,E2 -26671.238} C_VEL
LIN {X 0,Y 152.528,Z 487.404,A -85,B 0,C 180,E1 -26673.472,E2 -26673.472} C_VEL
LIN {X 0,Y 150.068,Z 515.239,A -85,B 0,C 180,E1 -26674.559,E2 -26674.559} C_VEL
LIN {X 0,Y 147.586,Z 529.08,A -85,B 0,C 180,E1 -26675.432,E2 -26675.432} C_VEL
LIN {X 0,Y 144.283,Z 541.114,A -85,B 0,C 180,E1 -26676.516,E2 -26676.516} C_VEL
LIN {X 0,Y 139.752,Z 553.766,A -85,B 0,C 180,E1 -26678.21,E2 -26678.21} C_VEL
LIN {X 0,Y 134.682,Z 565.024,A -85,B 0,C 180,E1 -26680.258,E2 -26680.258} C_VEL
LIN {X 0,Y 129.323,Z 575.171,A -85,B 0,C 180,E1 -26682.808,E2 -26682.808} C_VEL
LIN {X 0,Y 123.661,Z 584.319,A -85,B 0,C 180,E1 -26685.878,E2 -26685.878} C_VEL
LIN {X 0,Y 117.468,Z 593.244,A -85,B 0,C 180,E1 -26689.973,E2 -26689.973} C_VEL
LIN {X 0,Y 111.618,Z 600.954,A -85,B 0,C 180,E1 -26694.939,E2 -26694.939} C_VEL
LIN {X 0,Y 108.256,Z 605.299,A -85,B 0,C 180,E1 -26698.711,E2 -26698.711} C_VEL
LIN {X 0,Y 104.237,Z 610.023,A -85,B 0,C 180,E1 -26704.008,E2 -26704.008} C_VEL
LIN {X 0,Y 101.15,Z 613.638,A -85,B 0,C 180,E1 -26709.672,E2 -26709.672} C_VEL
LIN {X 0,Y 99.754,Z 615.509,A -85,B 0,C 180,E1 -26713.632,E2 -26713.632} C_VEL
LIN {X 0,Y 98.778,Z 616.916,A -85,B 0,C 180,E1 -26717.676,E2 -26717.676} C_VEL
LIN {X 0,Y 98.212,Z 617.925,A -85,B 0,C 180,E1 -26721.772,E2 -26721.772} C_VEL
LIN {X 0,Y 98.02,Z 618.544,A -85,B 0,C 180,E1 -26725.888,E2 -26725.888} C_VEL
LIN {X 0,Y 98.146,Z 618.764,A -85,B 0,C 180,E1 -26730,E2 -26730} C_VEL
LIN {X 0,Y 98.022,Z 618.527,A -85,B 0,C 180,E1 -26734.111,E2 -26734.111} C_VEL
LIN {X 0,Y 98.211,Z 617.897,A -85,B 0,C 180,E1 -26738.228,E2 -26738.228} C_VEL
LIN {X 0,Y 98.773,Z 616.877,A -85,B 0,C 180,E1 -26742.325,E2 -26742.325} C_VEL
LIN {X 0,Y 99.748,Z 615.452,A -85,B 0,C 180,E1 -26746.369,E2 -26746.369} C_VEL
LIN {X 0,Y 102.064,Z 612.48,A -85,B 0,C 180,E1 -26752.254,E2 -26752.254} C_VEL
LIN {X 0,Y 105.465,Z 608.475,A -85,B 0,C 180,E1 -26757.805,E2 -26757.805} C_VEL
LIN {X 0,Y 110.557,Z 602.326,A -85,B 0,C 180,E1 -26763.795,E2 -26763.795} C_VEL
LIN {X 0,Y 115.633,Z 595.614,A -85,B 0,C 180,E1 -26768.533,E2 -26768.533} C_VEL
LIN {X 0,Y 121.548,Z 587.304,A -85,B 0,C 180,E1 -26772.795,E2 -26772.795} C_VEL
LIN {X 0,Y 127.033,Z 578.784,A -85,B 0,C 180,E1 -26775.988,E2 -26775.988} C_VEL
LIN {X 0,Y 132.885,Z 568.264,A -85,B 0,C 180,E1 -26778.906,E2 -26778.906} C_VEL
LIN {X 0,Y 138.435,Z 556.421,A -85,B 0,C 180,E1 -26781.309,E2 -26781.309} C_VEL
LIN {X 0,Y 142.968,Z 544.481,A -85,B 0,C 180,E1 -26783.015,E2 -26783.015} C_VEL
LIN {X 0,Y 146.599,Z 532.047,A -85,B 0,C 180,E1 -26784.289,E2 -26784.289} C_VEL
LIN {X 0,Y 149.187,Z 519.597,A -85,B 0,C 180,E1 -26785.168,E2 -26785.168} C_VEL
LIN {X 0,Y 150.36,Z 510.79,A -85,B 0,C 180,E1 -26785.58,E2 -26785.58} C_VEL
LIN {X 0,Y 150.625,Z 504.973,A -85,B 0,C 180,E1 -26785.977,E2 -26785.977} C_VEL
LIN {X 0,Y 150.174,Z 499.375,A -85,B 0,C 180,E1 -26786.721,E2 -26786.721} C_VEL
LIN {X 0,Y 148.823,Z 492.347,A -85,B 0,C 180,E1 -26788.116,E2 -26788.116} C_VEL
LIN {X 0,Y 146.066,Z 482.644,A -85,B 0,C 180,E1 -26790.779,E2 -26790.779} C_VEL
LIN {X 0,Y 143.382,Z 475.238,A -85,B 0,C 180,E1 -26793.53,E2 -26793.53} C_VEL
LIN {X 0,Y 140.851,Z 469.264,A -85,B 0,C 180,E1 -26796.376,E2 -26796.376} C_VEL
LIN {X 0,Y 138.019,Z 464.31,A -85,B 0,C 180,E1 -26799.897,E2 -26799.897} C_VEL
LIN {X 0,Y 135.548,Z 460.357,A -85,B 0,C 180,E1 -26803.625,E2 -26803.625} C_VEL
LIN {X 0,Y 133.282,Z 456.479,A -85,B 0,C 180,E1 -26808.21,E2 -26808.21} C_VEL
LIN {X 0,Y 131.063,Z 452.362,A -85,B 0,C 180,E1 -26816.926,E2 -26816.926} C_VEL
LIN {X 0,Y 130.999,Z 451.588,A -85,B 0,C 180,E1 -26818.463,E2 -26818.463} C_VEL
LIN {X 0,Y 131.022,Z 451.799,A -85,B 0,C 180,E1 -26822.69,E2 -26822.69} C_VEL
LIN {X 0,Y 132.9,Z 456.174,A -85,B 0,C 180,E1 -26831.485,E2 -26831.485} C_VEL
LIN {X 0,Y 133.593,Z 457.067,A -85,B 0,C 180,E1 -26833.113,E2 -26833.113} C_VEL
LIN {X 0,Y 136.299,Z 461.56,A -85,B 0,C 180,E1 -26838.178,E2 -26838.178} C_VEL
LIN {X 0,Y 139.079,Z 466.166,A -85,B 0,C 180,E1 -26842.077,E2 -26842.077} C_VEL
LIN {X 0,Y 142.168,Z 471.512,A -85,B 0,C 180,E1 -26845.63,E2 -26845.63} C_VEL
LIN {X 0,Y 145.985,Z 478.905,A -85,B 0,C 180,E1 -26849.37,E2 -26849.37} C_VEL
LIN {X 0,Y 148.712,Z 484.967,A -85,B 0,C 180,E1 -26851.76,E2 -26851.76} C_VEL
LIN {X 0,Y 146.274,Z 509.829,A -85,B 0,C 180,E1 -26852.693,E2 -26852.693} C_VEL
LIN {X 0,Y 143.864,Z 522.858,A -85,B 0,C 180,E1 -26853.536,E2 -26853.536} C_VEL
LIN {X 0,Y 140.685,Z 535.092,A -85,B 0,C 180,E1 -26854.802,E2 -26854.802} C_VEL
LIN {X 0,Y 136.51,Z 546.857,A -85,B 0,C 180,E1 -26856.447,E2 -26856.447} C_VEL
LIN {X 0,Y 131.487,Z 558.169,A -85,B 0,C 180,E1 -26858.585,E2 -26858.585} C_VEL
LIN {X 0,Y 126.008,Z 568.362,A -85,B 0,C 180,E1 -26861.155,E2 -26861.155} C_VEL
LIN {X 0,Y 120.359,Z 577.502,A -85,B 0,C 180,E1 -26864.333,E2 -26864.333} C_VEL
LIN {X 0,Y 114.04,Z 586.386,A -85,B 0,C 180,E1 -26868.511,E2 -26868.511} C_VEL
LIN {X 0,Y 108.248,Z 593.536,A -85,B 0,C 180,E1 -26873.091,E2 -26873.091} C_VEL
LIN {X 0,Y 103.837,Z 598.359,A -85,B 0,C 180,E1 -26877.217,E2 -26877.217} C_VEL
LIN {X 0,Y 99.488,Z 603.034,A -85,B 0,C 180,E1 -26882.667,E2 -26882.667} C_VEL
LIN {X 0,Y 95.995,Z 606.608,A -85,B 0,C 180,E1 -26888.528,E2 -26888.528} C_VEL
LIN {X 0,Y 94.193,Z 608.451,A -85,B 0,C 180,E1 -26892.636,E2 -26892.636} C_VEL
LIN {X 0,Y 92.809,Z 609.833,A -85,B 0,C 180,E1 -26896.869,E2 -26896.869} C_VEL
LIN {X 0,Y 91.877,Z 610.814,A -85,B 0,C 180,E1 -26901.2,E2 -26901.2} C_VEL
LIN {X 0,Y 91.222,Z 611.638,A -85,B 0,C 180,E1 -26910,E2 -26910} C_VEL
LIN {X 0,Y 91.325,Z 611.444,A -85,B 0,C 180,E1 -26914.414,E2 -26914.414} C_VEL
LIN {X 0,Y 91.877,Z 610.859,A -85,B 0,C 180,E1 -26918.8,E2 -26918.8} C_VEL
LIN {X 0,Y 94.189,Z 608.54,A -85,B 0,C 180,E1 -26927.365,E2 -26927.365} C_VEL
LIN {X 0,Y 97.017,Z 605.678,A -85,B 0,C 180,E1 -26933.479,E2 -26933.479} C_VEL
LIN {X 0,Y 100.829,Z 601.791,A -85,B 0,C 180,E1 -26939.203,E2 -26939.203} C_VEL
LIN {X 0,Y 105.454,Z 596.775,A -85,B 0,C 180,E1 -26944.504,E2 -26944.504} C_VEL
LIN {X 0,Y 110.981,Z 590.444,A -85,B 0,C 180,E1 -26949.29,E2 -26949.29} C_VEL
LIN {X 0,Y 116.987,Z 582.568,A -85,B 0,C 180,E1 -26953.669,E2 -26953.669} C_VEL
LIN {X 0,Y 122.438,Z 574.465,A -85,B 0,C 180,E1 -26957.041,E2 -26957.041} C_VEL
LIN {X 0,Y 128.301,Z 564.612,A -85,B 0,C 180,E1 -26960.073,E2 -26960.073} C_VEL
LIN {X 0,Y 133.869,Z 553.502,A -85,B 0,C 180,E1 -26962.563,E2 -26962.563} C_VEL
LIN {X 0,Y 138.366,Z 542.607,A -85,B 0,C 180,E1 -26964.357,E2 -26964.357} C_VEL
LIN {X 0,Y 142.234,Z 530.561,A -85,B 0,C 180,E1 -26965.856,E2 -26965.856} C_VEL
LIN {X 0,Y 145.169,Z 518.146,A -85,B 0,C 180,E1 -26966.936,E2 -26966.936} C_VEL
LIN {X 0,Y 147.152,Z 504.702,A -85,B 0,C 180,E1 -26967.685,E2 -26967.685} C_VEL
LIN {X 0,Y 148.87,Z 484.985,A -85,B 0,C 180,E1 -26968.435,E2 -26968.435} C_VEL
LIN {X 0,Y 144.957,Z 476.607,A -85,B 0,C 180,E1 -26971.937,E2 -26971.937} C_VEL
LIN {X 0,Y 141.472,Z 470.156,A -85,B 0,C 180,E1 -26975.512,E2 -26975.512} C_VEL
LIN {X 0,Y 138.34,Z 464.66,A -85,B 0,C 180,E1 -26979.363,E2 -26979.363} C_VEL
LIN {X 0,Y 135.772,Z 460.527,A -85,B 0,C 180,E1 -26983.25,E2 -26983.25} C_VEL
LIN {X 0,Y 133.641,Z 456.845,A -85,B 0,C 180,E1 -26987.568,E2 -26987.568} C_VEL
LIN {X 0,Y 131.278,Z 451.581,A -85,B 0,C 180,E1 -26999.285,E2 -26999.285} C_VEL
LIN {X 0,Y 131.263,Z 452.04,A -85,B 0,C 180,E1 -27001.261,E2 -27001.261} C_VEL
LIN {X 0,Y 133.716,Z 457.008,A -85,B 0,C 180,E1 -27012.136,E2 -27012.136} C_VEL
LIN {X 0,Y 135.8,Z 460.544,A -85,B 0,C 180,E1 -27016.309,E2 -27016.309} C_VEL
LIN {X 0,Y 138.921,Z 465.704,A -85,B 0,C 180,E1 -27020.934,E2 -27020.934} C_VEL
LIN {X 0,Y 141.393,Z 470.032,A -85,B 0,C 180,E1 -27023.917,E2 -27023.917} C_VEL
LIN {X 0,Y 144.388,Z 477.479,A -85,B 0,C 180,E1 -27027.24,E2 -27027.24} C_VEL
LIN {X 0,Y 147.397,Z 486.198,A -85,B 0,C 180,E1 -27030.24,E2 -27030.24} C_VEL
LIN {X 0,Y 148.495,Z 489.729,A -85,B 0,C 180,E1 -27031.274,E2 -27031.274} C_VEL
LIN {X 0,Y 146.069,Z 515.605,A -85,B 0,C 180,E1 -27032.299,E2 -27032.299} C_VEL
LIN {X 0,Y 143.488,Z 529.275,A -85,B 0,C 180,E1 -27033.158,E2 -27033.158} C_VEL
LIN {X 0,Y 140.18,Z 540.854,A -85,B 0,C 180,E1 -27034.186,E2 -27034.186} C_VEL
LIN {X 0,Y 135.466,Z 553.503,A -85,B 0,C 180,E1 -27035.845,E2 -27035.845} C_VEL
LIN {X 0,Y 130.211,Z 564.761,A -85,B 0,C 180,E1 -27037.875,E2 -27037.875} C_VEL
LIN {X 0,Y 124.603,Z 574.907,A -85,B 0,C 180,E1 -27040.41,E2 -27040.41} C_VEL
LIN {X 0,Y 118.648,Z 584.053,A -85,B 0,C 180,E1 -27043.481,E2 -27043.481} C_VEL
LIN {X 0,Y 112.094,Z 592.978,A -85,B 0,C 180,E1 -27047.625,E2 -27047.625} C_VEL
LIN {X 0,Y 106.332,Z 600.167,A -85,B 0,C 180,E1 -27052.312,E2 -27052.312} C_VEL
LIN {X 0,Y 102.24,Z 605.032,A -85,B 0,C 180,E1 -27056.639,E2 -27056.639} C_VEL
LIN {X 0,Y 97.878,Z 609.755,A -85,B 0,C 180,E1 -27062.179,E2 -27062.179} C_VEL
LIN {X 0,Y 94.486,Z 613.37,A -85,B 0,C 180,E1 -27068.167,E2 -27068.167} C_VEL
LIN {X 0,Y 92.931,Z 615.241,A -85,B 0,C 180,E1 -27072.392,E2 -27072.392} C_VEL
LIN {X 0,Y 91.828,Z 616.648,A -85,B 0,C 180,E1 -27076.727,E2 -27076.727} C_VEL
LIN {X 0,Y 91.163,Z 617.657,A -85,B 0,C 180,E1 -27081.131,E2 -27081.131} C_VEL
LIN {X 0,Y 90.927,Z 618.277,A -85,B 0,C 180,E1 -27085.567,E2 -27085.567} C_VEL
LIN {X 0,Y 91.049,Z 618.497,A -85,B 0,C 180,E1 -27090,E2 -27090} C_VEL
LIN {X 0,Y 90.928,Z 618.259,A -85,B 0,C 180,E1 -27094.433,E2 -27094.433} C_VEL
LIN {X 0,Y 91.162,Z 617.628,A -85,B 0,C 180,E1 -27098.869,E2 -27098.869} C_VEL
LIN {X 0,Y 91.823,Z 616.608,A -85,B 0,C 180,E1 -27103.274,E2 -27103.274} C_VEL
LIN {X 0,Y 92.926,Z 615.183,A -85,B 0,C 180,E1 -27107.609,E2 -27107.609} C_VEL
LIN {X 0,Y 95.501,Z 612.21,A -85,B 0,C 180,E1 -27113.875,E2 -27113.875} C_VEL
LIN {X 0,Y 99.197,Z 608.205,A -85,B 0,C 180,E1 -27119.731,E2 -27119.731} C_VEL
LIN {X 0,Y 104.675,Z 602.055,A -85,B 0,C 180,E1 -27125.978,E2 -27125.978} C_VEL
LIN {X 0,Y 110.128,Z 595.343,A -85,B 0,C 180,E1 -27130.852,E2 -27130.852} C_VEL
LIN {X 0,Y 116.412,Z 587.033,A -85,B 0,C 180,E1 -27135.182,E2 -27135.182} C_VEL
LIN {X 0,Y 122.2,Z 578.514,A -85,B 0,C 180,E1 -27138.387,E2 -27138.387} C_VEL
LIN {X 0,Y 128.324,Z 567.993,A -85,B 0,C 180,E1 -27141.299,E2 -27141.299} C_VEL
LIN {X 0,Y 134.111,Z 556.149,A -85,B 0,C 180,E1 -27143.678,E2 -27143.678} C_VEL
LIN {X 0,Y 138.815,Z 544.208,A -85,B 0,C 180,E1 -27145.356,E2 -27145.356} C_VEL
LIN {X 0,Y 142.573,Z 531.772,A -85,B 0,C 180,E1 -27146.605,E2 -27146.605} C_VEL
LIN {X 0,Y 145.276,Z 519.227,A -85,B 0,C 180,E1 -27147.466,E2 -27147.466} C_VEL
LIN {X 0,Y 147.011,Z 504.954,A -85,B 0,C 180,E1 -27148.073,E2 -27148.073} C_VEL
LIN {X 0,Y 148.301,Z 489.593,A -85,B 0,C 180,E1 -27148.653,E2 -27148.653} C_VEL
LIN {X 0,Y 146.066,Z 482.644,A -85,B 0,C 180,E1 -27150.779,E2 -27150.779} C_VEL
LIN {X 0,Y 144.986,Z 479.935,A -85,B 0,C 180,E1 -27151.817,E2 -27151.817} C_VEL
LIN {X 0,Y 142.987,Z 476.85,A -85,B 0,C 180,E1 -27153.668,E2 -27153.668} C_VEL
LIN {X 0,Y 140.832,Z 474.65,A -85,B 0,C 180,E1 -27155.738,E2 -27155.738} C_VEL
LIN {X 0,Y 135.63,Z 469.767,A -85,B 0,C 180,E1 -27161.893,E2 -27161.893} C_VEL
LIN {X 0,Y 134.038,Z 466.921,A -85,B 0,C 180,E1 -27164.607,E2 -27164.607} C_VEL
LIN {X 0,Y 132.1,Z 463.334,A -85,B 0,C 180,E1 -27168.88,E2 -27168.88} C_VEL
LIN {X 0,Y 130.096,Z 458.582,A -85,B 0,C 180,E1 -27179.226,E2 -27179.226} C_VEL
LIN {X 0,Y 130.125,Z 458.837,A -85,B 0,C 180,E1 -27182.322,E2 -27182.322} C_VEL
LIN {X 0,Y 131.886,Z 463.154,A -85,B 0,C 180,E1 -27191.174,E2 -27191.174} C_VEL
LIN {X 0,Y 132.441,Z 464.1,A -85,B 0,C 180,E1 -27192.597,E2 -27192.597} C_VEL
LIN {X 0,Y 134.789,Z 468.221,A -85,B 0,C 180,E1 -27197.3,E2 -27197.3} C_VEL
LIN {X 0,Y 137.235,Z 472.551,A -85,B 0,C 180,E1 -27201.007,E2 -27201.007} C_VEL
LIN {X 0,Y 140.087,Z 477.798,A -85,B 0,C 180,E1 -27204.549,E2 -27204.549} C_VEL
LIN {X 0,Y 143.501,Z 484.927,A -85,B 0,C 180,E1 -27208.172,E2 -27208.172} C_VEL
LIN {X 0,Y 144.862,Z 488.178,A -85,B 0,C 180,E1 -27209.498,E2 -27209.498} C_VEL
LIN {X 0,Y 142.63,Z 509.728,A -85,B 0,C 180,E1 -27210.278,E2 -27210.278} C_VEL
LIN {X 0,Y 140.13,Z 522.873,A -85,B 0,C 180,E1 -27211.098,E2 -27211.098} C_VEL
LIN {X 0,Y 136.768,Z 535.365,A -85,B 0,C 180,E1 -27212.366,E2 -27212.366} C_VEL
LIN {X 0,Y 132.419,Z 547.129,A -85,B 0,C 180,E1 -27213.977,E2 -27213.977} C_VEL
LIN {X 0,Y 127.188,Z 558.44,A -85,B 0,C 180,E1 -27216.088,E2 -27216.088} C_VEL
LIN {X 0,Y 121.465,Z 568.631,A -85,B 0,C 180,E1 -27218.639,E2 -27218.639} C_VEL
LIN {X 0,Y 115.511,Z 577.772,A -85,B 0,C 180,E1 -27221.815,E2 -27221.815} C_VEL
LIN {X 0,Y 108.816,Z 586.655,A -85,B 0,C 180,E1 -27226.03,E2 -27226.03} C_VEL
LIN {X 0,Y 102.674,Z 593.804,A -85,B 0,C 180,E1 -27230.717,E2 -27230.717} C_VEL
LIN {X 0,Y 97.94,Z 598.628,A -85,B 0,C 180,E1 -27234.967,E2 -27234.967} C_VEL
LIN {X 0,Y 93.236,Z 603.303,A -85,B 0,C 180,E1 -27240.663,E2 -27240.663} C_VEL
LIN {X 0,Y 89.431,Z 606.876,A -85,B 0,C 180,E1 -27246.864,E2 -27246.864} C_VEL
LIN {X 0,Y 87.439,Z 608.719,A -85,B 0,C 180,E1 -27251.247,E2 -27251.247} C_VEL
LIN {X 0,Y 84.874,Z 611.082,A -85,B 0,C 180,E1 -27260.468,E2 -27260.468} C_VEL
LIN {X 0,Y 84.141,Z 611.905,A -85,B 0,C 180,E1 -27270,E2 -27270} C_VEL
LIN {X 0,Y 84.264,Z 611.71,A -85,B 0,C 180,E1 -27274.784,E2 -27274.784} C_VEL
LIN {X 0,Y 84.874,Z 611.126,A -85,B 0,C 180,E1 -27279.532,E2 -27279.532} C_VEL
LIN {X 0,Y 87.433,Z 608.807,A -85,B 0,C 180,E1 -27288.755,E2 -27288.755} C_VEL
LIN {X 0,Y 90.541,Z 605.945,A -85,B 0,C 180,E1 -27295.272,E2 -27295.272} C_VEL
LIN {X 0,Y 94.678,Z 602.057,A -85,B 0,C 180,E1 -27301.305,E2 -27301.305} C_VEL
LIN {X 0,Y 99.687,Z 597.04,A -85,B 0,C 180,E1 -27306.815,E2 -27306.815} C_VEL
LIN {X 0,Y 105.582,Z 590.71,A -85,B 0,C 180,E1 -27311.731,E2 -27311.731} C_VEL
LIN {X 0,Y 111.598,Z 583.312,A -85,B 0,C 180,E1 -27315.949,E2 -27315.949} C_VEL
LIN {X 0,Y 117.708,Z 574.73,A -85,B 0,C 180,E1 -27319.574,E2 -27319.574} C_VEL
LIN {X 0,Y 123.868,Z 564.875,A -85,B 0,C 180,E1 -27322.59,E2 -27322.59} C_VEL
LIN {X 0,Y 129.677,Z 553.764,A -85,B 0,C 180,E1 -27325.054,E2 -27325.054} C_VEL
LIN {X 0,Y 134.368,Z 542.868,A -85,B 0,C 180,E1 -27326.809,E2 -27326.809} C_VEL
LIN {X 0,Y 138.379,Z 530.82,A -85,B 0,C 180,E1 -27328.286,E2 -27328.286} C_VEL
LIN {X 0,Y 141.391,Z 518.612,A -85,B 0,C 180,E1 -27329.326,E2 -27329.326} C_VEL
LIN {X 0,Y 143.495,Z 504.871,A -85,B 0,C 180,E1 -27330.083,E2 -27330.083} C_VEL
LIN {X 0,Y 145.02,Z 488.146,A -85,B 0,C 180,E1 -27330.715,E2 -27330.715} C_VEL
LIN {X 0,Y 141.761,Z 480.93,A -85,B 0,C 180,E1 -27333.995,E2 -27333.995} C_VEL
LIN {X 0,Y 138.346,Z 474.226,A -85,B 0,C 180,E1 -27338.004,E2 -27338.004} C_VEL
LIN {X 0,Y 135.958,Z 470.117,A -85,B 0,C 180,E1 -27341.346,E2 -27341.346} C_VEL
LIN {X 0,Y 134.181,Z 466.985,A -85,B 0,C 180,E1 -27344.39,E2 -27344.39} C_VEL
LIN {X 0,Y 132.2,Z 463.357,A -85,B 0,C 180,E1 -27348.889,E2 -27348.889} C_VEL
LIN {X 0,Y 130.403,Z 458.711,A -85,B 0,C 180,E1 -27359.28,E2 -27359.28} C_VEL
LIN {X 0,Y 130.382,Z 459.022,A -85,B 0,C 180,E1 -27360.793,E2 -27360.793} C_VEL
LIN {X 0,Y 132.452,Z 463.739,A -85,B 0,C 180,E1 -27371.283,E2 -27371.283} C_VEL
LIN {X 0,Y 134.821,Z 468.08,A -85,B 0,C 180,E1 -27376.288,E2 -27376.288} C_VEL
LIN {X 0,Y 137.356,Z 472.525,A -85,B 0,C 180,E1 -27380.204,E2 -27380.204} C_VEL
LIN {X 0,Y 139.285,Z 476.262,A -85,B 0,C 180,E1 -27382.725,E2 -27382.725} C_VEL
LIN {X 0,Y 142.025,Z 483.696,A -85,B 0,C 180,E1 -27386.051,E2 -27386.051} C_VEL
LIN {X 0,Y 144.689,Z 492.302,A -85,B 0,C 180,E1 -27388.98,E2 -27388.98} C_VEL
LIN {X 0,Y 142.392,Z 515.351,A -85,B 0,C 180,E1 -27389.877,E2 -27389.877} C_VEL
LIN {X 0,Y 139.719,Z 529.082,A -85,B 0,C 180,E1 -27390.726,E2 -27390.726} C_VEL
LIN {X 0,Y 136.324,Z 540.593,A -85,B 0,C 180,E1 -27391.721,E2 -27391.721} C_VEL
LIN {X 0,Y 131.435,Z 553.241,A -85,B 0,C 180,E1 -27393.336,E2 -27393.336} C_VEL
LIN {X 0,Y 125.985,Z 564.499,A -85,B 0,C 180,E1 -27395.331,E2 -27395.331} C_VEL
LIN {X 0,Y 120.113,Z 574.642,A -85,B 0,C 180,E1 -27397.825,E2 -27397.825} C_VEL
LIN {X 0,Y 113.867,Z 583.788,A -85,B 0,C 180,E1 -27400.882,E2 -27400.882} C_VEL
LIN {X 0,Y 106.928,Z 592.711,A -85,B 0,C 180,E1 -27405.046,E2 -27405.046} C_VEL
LIN {X 0,Y 100.772,Z 599.9,A -85,B 0,C 180,E1 -27409.827,E2 -27409.827} C_VEL
LIN {X 0,Y 96.363,Z 604.766,A -85,B 0,C 180,E1 -27414.307,E2 -27414.307} C_VEL
LIN {X 0,Y 91.633,Z 609.488,A -85,B 0,C 180,E1 -27420.098,E2 -27420.098} C_VEL
LIN {X 0,Y 87.898,Z 613.102,A -85,B 0,C 180,E1 -27426.436,E2 -27426.436} C_VEL
LIN {X 0,Y 86.166,Z 614.973,A -85,B 0,C 180,E1 -27430.959,E2 -27430.959} C_VEL
LIN {X 0,Y 84.916,Z 616.381,A -85,B 0,C 180,E1 -27435.624,E2 -27435.624} C_VEL
LIN {X 0,Y 83.857,Z 618.01,A -85,B 0,C 180,E1 -27445.193,E2 -27445.193} C_VEL
LIN {X 0,Y 83.946,Z 618.23,A -85,B 0,C 180,E1 -27450,E2 -27450} C_VEL
LIN {X 0,Y 83.857,Z 617.992,A -85,B 0,C 180,E1 -27454.807,E2 -27454.807} C_VEL
LIN {X 0,Y 84.912,Z 616.34,A -85,B 0,C 180,E1 -27464.377,E2 -27464.377} C_VEL
LIN {X 0,Y 86.162,Z 614.914,A -85,B 0,C 180,E1 -27469.042,E2 -27469.042} C_VEL
LIN {X 0,Y 89.029,Z 611.941,A -85,B 0,C 180,E1 -27475.732,E2 -27475.732} C_VEL
LIN {X 0,Y 93.061,Z 607.935,A -85,B 0,C 180,E1 -27481.913,E2 -27481.913} C_VEL
LIN {X 0,Y 98.055,Z 602.844,A -85,B 0,C 180,E1 -27487.461,E2 -27487.461} C_VEL
LIN {X 0,Y 103.816,Z 596.313,A -85,B 0,C 180,E1 -27492.606,E2 -27492.606} C_VEL
LIN {X 0,Y 110.352,Z 588.255,A -85,B 0,C 180,E1 -27497.087,E2 -27497.087} C_VEL
LIN {X 0,Y 116.349,Z 580.051,A -85,B 0,C 180,E1 -27500.367,E2 -27500.367} C_VEL
LIN {X 0,Y 122.674,Z 570.048,A -85,B 0,C 180,E1 -27503.326,E2 -27503.326} C_VEL
LIN {X 0,Y 128.692,Z 558.741,A -85,B 0,C 180,E1 -27505.687,E2 -27505.687} C_VEL
LIN {X 0,Y 133.483,Z 547.659,A -85,B 0,C 180,E1 -27507.394,E2 -27507.394} C_VEL
LIN {X 0,Y 137.743,Z 535.36,A -85,B 0,C 180,E1 -27508.717,E2 -27508.717} C_VEL
LIN {X 0,Y 140.88,Z 522.663,A -85,B 0,C 180,E1 -27509.663,E2 -27509.663} C_VEL
LIN {X 0,Y 142.84,Z 510.063,A -85,B 0,C 180,E1 -27510.285,E2 -27510.285} C_VEL
LIN {X 0,Y 144.446,Z 492.056,A -85,B 0,C 180,E1 -27510.985,E2 -27510.985} C_VEL
LIN {X 0,Y 141.716,Z 483.245,A -85,B 0,C 180,E1 -27513.987,E2 -27513.987} C_VEL
LIN {X 0,Y 138.838,Z 475.518,A -85,B 0,C 180,E1 -27517.492,E2 -27517.492} C_VEL
LIN {X 0,Y 136.115,Z 470.5,A -85,B 0,C 180,E1 -27521.173,E2 -27521.173} C_VEL
LIN {X 0,Y 135.63,Z 469.767,A -85,B 0,C 180,E1 -27521.893,E2 -27521.893} C_VEL
LIN {X 0,Y 134.109,Z 468.29,A -85,B 0,C 180,E1 -27524.237,E2 -27524.237} C_VEL
LIN {X 0,Y 132.635,Z 467.901,A -85,B 0,C 180,E1 -27526.712,E2 -27526.712} C_VEL
LIN {X 0,Y 129.782,Z 468.098,A -85,B 0,C 180,E1 -27533.627,E2 -27533.627} C_VEL
LIN {X 0,Y 129.449,Z 467.542,A -85,B 0,C 180,E1 -27535.378,E2 -27535.378} C_VEL
LIN {X 0,Y 129.227,Z 465.66,A -85,B 0,C 180,E1 -27539.221,E2 -27539.221} C_VEL
LIN {X 0,Y 129.234,Z 465.865,A -85,B 0,C 180,E1 -27541.948,E2 -27541.948} C_VEL
LIN {X 0,Y 130.704,Z 469.992,A -85,B 0,C 180,E1 -27550.402,E2 -27550.402} C_VEL
LIN {X 0,Y 131.409,Z 471.349,A -85,B 0,C 180,E1 -27552.353,E2 -27552.353} C_VEL
LIN {X 0,Y 133.343,Z 474.923,A -85,B 0,C 180,E1 -27556.457,E2 -27556.457} C_VEL
LIN {X 0,Y 135.374,Z 478.759,A -85,B 0,C 180,E1 -27559.804,E2 -27559.804} C_VEL
LIN {X 0,Y 138.332,Z 484.733,A -85,B 0,C 180,E1 -27563.783,E2 -27563.783} C_VEL
LIN {X 0,Y 141.007,Z 490.814,A -85,B 0,C 180,E1 -27566.856,E2 -27566.856} C_VEL
LIN {X 0,Y 141.164,Z 491.206,A -85,B 0,C 180,E1 -27567.027,E2 -27567.027} C_VEL
LIN {X 0,Y 139.122,Z 510.462,A -85,B 0,C 180,E1 -27567.78,E2 -27567.78} C_VEL
LIN {X 0,Y 136.436,Z 523.87,A -85,B 0,C 180,E1 -27568.604,E2 -27568.604} C_VEL
LIN {X 0,Y 132.744,Z 536.631,A -85,B 0,C 180,E1 -27569.896,E2 -27569.896} C_VEL
LIN {X 0,Y 128.592,Z 547.401,A -85,B 0,C 180,E1 -27571.357,E2 -27571.357} C_VEL
LIN {X 0,Y 123.138,Z 558.711,A -85,B 0,C 180,E1 -27573.417,E2 -27573.417} C_VEL
LIN {X 0,Y 117.169,Z 568.901,A -85,B 0,C 180,E1 -27575.93,E2 -27575.93} C_VEL
LIN {X 0,Y 110.901,Z 578.042,A -85,B 0,C 180,E1 -27579.078,E2 -27579.078} C_VEL
LIN {X 0,Y 103.817,Z 586.925,A -85,B 0,C 180,E1 -27583.305,E2 -27583.305} C_VEL
LIN {X 0,Y 97.29,Z 594.073,A -85,B 0,C 180,E1 -27588.073,E2 -27588.073} C_VEL
LIN {X 0,Y 92.218,Z 598.896,A -85,B 0,C 180,E1 -27592.434,E2 -27592.434} C_VEL
LIN {X 0,Y 87.117,Z 603.571,A -85,B 0,C 180,E1 -27598.375,E2 -27598.375} C_VEL
LIN {X 0,Y 82.958,Z 607.143,A -85,B 0,C 180,E1 -27604.939,E2 -27604.939} C_VEL
LIN {X 0,Y 80.755,Z 608.986,A -85,B 0,C 180,E1 -27609.629,E2 -27609.629} C_VEL
LIN {X 0,Y 77.878,Z 611.349,A -85,B 0,C 180,E1 -27619.602,E2 -27619.602} C_VEL
LIN {X 0,Y 77.061,Z 612.171,A -85,B 0,C 180,E1 -27630,E2 -27630} C_VEL
LIN {X 0,Y 77.211,Z 611.977,A -85,B 0,C 180,E1 -27635.222,E2 -27635.222} C_VEL
LIN {X 0,Y 79.045,Z 610.429,A -85,B 0,C 180,E1 -27645.47,E2 -27645.47} C_VEL
LIN {X 0,Y 80.748,Z 609.073,A -85,B 0,C 180,E1 -27650.373,E2 -27650.373} C_VEL
LIN {X 0,Y 84.172,Z 606.211,A -85,B 0,C 180,E1 -27657.336,E2 -27657.336} C_VEL
LIN {X 0,Y 88.672,Z 602.324,A -85,B 0,C 180,E1 -27663.696,E2 -27663.696} C_VEL
LIN {X 0,Y 94.107,Z 597.305,A -85,B 0,C 180,E1 -27669.403,E2 -27669.403} C_VEL
LIN {X 0,Y 100.395,Z 590.975,A -85,B 0,C 180,E1 -27674.428,E2 -27674.428} C_VEL
LIN {X 0,Y 106.415,Z 584.043,A -85,B 0,C 180,E1 -27678.462,E2 -27678.462} C_VEL
LIN {X 0,Y 113.236,Z 574.994,A -85,B 0,C 180,E1 -27682.308,E2 -27682.308} C_VEL
LIN {X 0,Y 119.7,Z 565.138,A -85,B 0,C 180,E1 -27685.282,E2 -27685.282} C_VEL
LIN {X 0,Y 125.754,Z 554.026,A -85,B 0,C 180,E1 -27687.701,E2 -27687.701} C_VEL
LIN {X 0,Y 130.618,Z 543.129,A -85,B 0,C 180,E1 -27689.415,E2 -27689.415} C_VEL
LIN {X 0,Y 134.791,Z 531.079,A -85,B 0,C 180,E1 -27690.847,E2 -27690.847} C_VEL
LIN {X 0,Y 137.915,Z 518.867,A -85,B 0,C 180,E1 -27691.856,E2 -27691.856} C_VEL
LIN {X 0,Y 140.03,Z 505.65,A -85,B 0,C 180,E1 -27692.578,E2 -27692.578} C_VEL
LIN {X 0,Y 141.393,Z 491.337,A -85,B 0,C 180,E1 -27693.127,E2 -27693.127} C_VEL
LIN {X 0,Y 138.371,Z 484.474,A -85,B 0,C 180,E1 -27696.614,E2 -27696.614} C_VEL
LIN {X 0,Y 135.406,Z 478.517,A -85,B 0,C 180,E1 -27700.677,E2 -27700.677} C_VEL
LIN {X 0,Y 132.798,Z 473.685,A -85,B 0,C 180,E1 -27705.245,E2 -27705.245} C_VEL
LIN {X 0,Y 131.054,Z 470.198,A -85,B 0,C 180,E1 -27709.572,E2 -27709.572} C_VEL
LIN {X 0,Y 129.524,Z 465.839,A -85,B 0,C 180,E1 -27720,E2 -27720} C_VEL
LIN {X 0,Y 131.28,Z 470.633,A -85,B 0,C 180,E1 -27730.604,E2 -27730.604} C_VEL
LIN {X 0,Y 133.402,Z 474.813,A -85,B 0,C 180,E1 -27735.463,E2 -27735.463} C_VEL
LIN {X 0,Y 135.635,Z 478.988,A -85,B 0,C 180,E1 -27739.19,E2 -27739.19} C_VEL
LIN {X 0,Y 137.241,Z 482.483,A -85,B 0,C 180,E1 -27741.498,E2 -27741.498} C_VEL
LIN {X 0,Y 139.673,Z 489.898,A -85,B 0,C 180,E1 -27744.775,E2 -27744.775} C_VEL
LIN {X 0,Y 141.116,Z 494.967,A -85,B 0,C 180,E1 -27746.568,E2 -27746.568} C_VEL
LIN {X 0,Y 138.964,Z 515.307,A -85,B 0,C 180,E1 -27747.352,E2 -27747.352} C_VEL
LIN {X 0,Y 136.226,Z 528.819,A -85,B 0,C 180,E1 -27748.155,E2 -27748.155} C_VEL
LIN {X 0,Y 132.736,Z 540.333,A -85,B 0,C 180,E1 -27749.119,E2 -27749.119} C_VEL
LIN {X 0,Y 127.675,Z 552.979,A -85,B 0,C 180,E1 -27750.675,E2 -27750.675} C_VEL
LIN {X 0,Y 122.018,Z 564.236,A -85,B 0,C 180,E1 -27752.611,E2 -27752.611} C_VEL
LIN {X 0,Y 115.868,Z 574.376,A -85,B 0,C 180,E1 -27755.033,E2 -27755.033} C_VEL
LIN {X 0,Y 109.336,Z 583.522,A -85,B 0,C 180,E1 -27758.057,E2 -27758.057} C_VEL
LIN {X 0,Y 102.017,Z 592.446,A -85,B 0,C 180,E1 -27762.221,E2 -27762.221} C_VEL
LIN {X 0,Y 95.431,Z 599.633,A -85,B 0,C 180,E1 -27767.063,E2 -27767.063} C_VEL
LIN {X 0,Y 88.83,Z 606.192,A -85,B 0,C 180,E1 -27773.604,E2 -27773.604} C_VEL
LIN {X 0,Y 84.038,Z 610.532,A -85,B 0,C 180,E1 -27779.883,E2 -27779.883} C_VEL
LIN {X 0,Y 81.409,Z 612.834,A -85,B 0,C 180,E1 -27784.428,E2 -27784.428} C_VEL
LIN {X 0,Y 79.451,Z 614.705,A -85,B 0,C 180,E1 -27789.279,E2 -27789.279} C_VEL
LIN {X 0,Y 78.021,Z 616.112,A -85,B 0,C 180,E1 -27794.322,E2 -27794.322} C_VEL
LIN {X 0,Y 76.776,Z 617.743,A -85,B 0,C 180,E1 -27804.748,E2 -27804.748} C_VEL
LIN {X 0,Y 76.852,Z 617.963,A -85,B 0,C 180,E1 -27810,E2 -27810} C_VEL
LIN {X 0,Y 76.776,Z 617.724,A -85,B 0,C 180,E1 -27815.252,E2 -27815.252} C_VEL
LIN {X 0,Y 78.017,Z 616.071,A -85,B 0,C 180,E1 -27825.679,E2 -27825.679} C_VEL
LIN {X 0,Y 79.447,Z 614.645,A -85,B 0,C 180,E1 -27830.722,E2 -27830.722} C_VEL
LIN {X 0,Y 82.669,Z 611.672,A -85,B 0,C 180,E1 -27837.876,E2 -27837.876} C_VEL
LIN {X 0,Y 87.085,Z 607.665,A -85,B 0,C 180,E1 -27844.396,E2 -27844.396} C_VEL
LIN {X 0,Y 92.953,Z 602.051,A -85,B 0,C 180,E1 -27850.658,E2 -27850.658} C_VEL
LIN {X 0,Y 99.76,Z 594.802,A -85,B 0,C 180,E1 -27856.227,E2 -27856.227} C_VEL
LIN {X 0,Y 106.849,Z 586.492,A -85,B 0,C 180,E1 -27860.61,E2 -27860.61} C_VEL
LIN {X 0,Y 113.233,Z 577.971,A -85,B 0,C 180,E1 -27863.789,E2 -27863.789} C_VEL
LIN {X 0,Y 119.939,Z 567.45,A -85,B 0,C 180,E1 -27866.614,E2 -27866.614} C_VEL
LIN {X 0,Y 126.225,Z 555.606,A -85,B 0,C 180,E1 -27868.874,E2 -27868.874} C_VEL
LIN {X 0,Y 131.26,Z 543.66,A -85,B 0,C 180,E1 -27870.464,E2 -27870.464} C_VEL
LIN {X 0,Y 135.286,Z 531.222,A -85,B 0,C 180,E1 -27871.627,E2 -27871.627} C_VEL
LIN {X 0,Y 138.249,Z 518.136,A -85,B 0,C 180,E1 -27872.466,E2 -27872.466} C_VEL
LIN {X 0,Y 140.206,Z 502.479,A -85,B 0,C 180,E1 -27873.072,E2 -27873.072} C_VEL
LIN {X 0,Y 140.862,Z 494.572,A -85,B 0,C 180,E1 -27873.418,E2 -27873.418} C_VEL
LIN {X 0,Y 138.592,Z 486.973,A -85,B 0,C 180,E1 -27876.265,E2 -27876.265} C_VEL
LIN {X 0,Y 136.555,Z 481.107,A -85,B 0,C 180,E1 -27879.081,E2 -27879.081} C_VEL
LIN {X 0,Y 134.393,Z 476.876,A -85,B 0,C 180,E1 -27882.304,E2 -27882.304} C_VEL
LIN {X 0,Y 132.476,Z 473.343,A -85,B 0,C 180,E1 -27885.797,E2 -27885.797} C_VEL
LIN {X 0,Y 130.824,Z 470.108,A -85,B 0,C 180,E1 -27889.847,E2 -27889.847} C_VEL
LIN {X 0,Y 129.449,Z 467.542,A -85,B 0,C 180,E1 -27895.378,E2 -27895.378} C_VEL
LIN {X 0,Y 129.207,Z 467.272,A -85,B 0,C 180,E1 -27897.098,E2 -27897.098} C_VEL
LIN {X 0,Y 128.979,Z 467.844,A -85,B 0,C 180,E1 -27898.817,E2 -27898.817} C_VEL
LIN {X 0,Y 128.674,Z 470.542,A -85,B 0,C 180,E1 -27902.152,E2 -27902.152} C_VEL
LIN {X 0,Y 128.933,Z 475.517,A -85,B 0,C 180,E1 -27907.203,E2 -27907.203} C_VEL
LIN {X 0,Y 129.348,Z 476.537,A -85,B 0,C 180,E1 -27908.959,E2 -27908.959} C_VEL
LIN {X 0,Y 129.998,Z 477.666,A -85,B 0,C 180,E1 -27911.004,E2 -27911.004} C_VEL
LIN {X 0,Y 131.855,Z 481.496,A -85,B 0,C 180,E1 -27915.457,E2 -27915.457} C_VEL
LIN {X 0,Y 134.008,Z 485.889,A -85,B 0,C 180,E1 -27919.269,E2 -27919.269} C_VEL
LIN {X 0,Y 136.794,Z 492.046,A -85,B 0,C 180,E1 -27923.238,E2 -27923.238} C_VEL
LIN {X 0,Y 137.808,Z 494.539,A -85,B 0,C 180,E1 -27924.526,E2 -27924.526} C_VEL
LIN {X 0,Y 135.874,Z 511.317,A -85,B 0,C 180,E1 -27925.167,E2 -27925.167} C_VEL
LIN {X 0,Y 133.245,Z 523.9,A -85,B 0,C 180,E1 -27925.907,E2 -27925.907} C_VEL
LIN {X 0,Y 129.74,Z 535.91,A -85,B 0,C 180,E1 -27927.077,E2 -27927.077} C_VEL
LIN {X 0,Y 125.767,Z 546.094,A -85,B 0,C 180,E1 -27928.345,E2 -27928.345} C_VEL
LIN {X 0,Y 120.077,Z 557.696,A -85,B 0,C 180,E1 -27930.313,E2 -27930.313} C_VEL
LIN {X 0,Y 113.825,Z 568.12,A -85,B 0,C 180,E1 -27932.729,E2 -27932.729} C_VEL
LIN {X 0,Y 107.856,Z 576.631,A -85,B 0,C 180,E1 -27935.463,E2 -27935.463} C_VEL
LIN {X 0,Y 101.303,Z 584.758,A -85,B 0,C 180,E1 -27939.013,E2 -27939.013} C_VEL
LIN {X 0,Y 94.377,Z 592.126,A -85,B 0,C 180,E1 -27943.445,E2 -27943.445} C_VEL
LIN {X 0,Y 86.702,Z 599.165,A -85,B 0,C 180,E1 -27949.575,E2 -27949.575} C_VEL
LIN {X 0,Y 81.16,Z 603.839,A -85,B 0,C 180,E1 -27955.747,E2 -27955.747} C_VEL
LIN {X 0,Y 76.569,Z 607.412,A -85,B 0,C 180,E1 -27962.683,E2 -27962.683} C_VEL
LIN {X 0,Y 74.133,Z 609.254,A -85,B 0,C 180,E1 -27967.716,E2 -27967.716} C_VEL
LIN {X 0,Y 72.246,Z 610.635,A -85,B 0,C 180,E1 -27973.032,E2 -27973.032} C_VEL
LIN {X 0,Y 70.162,Z 612.217,A -85,B 0,C 180,E1 -27984.251,E2 -27984.251} C_VEL
LIN {X 0,Y 69.969,Z 612.438,A -85,B 0,C 180,E1 -27990,E2 -27990} C_VEL
LIN {X 0,Y 70.162,Z 612.243,A -85,B 0,C 180,E1 -27995.749,E2 -27995.749} C_VEL
LIN {X 0,Y 72.245,Z 610.695,A -85,B 0,C 180,E1 -28006.968,E2 -28006.968} C_VEL
LIN {X 0,Y 74.125,Z 609.34,A -85,B 0,C 180,E1 -28012.287,E2 -28012.287} C_VEL
LIN {X 0,Y 77.937,Z 606.478,A -85,B 0,C 180,E1 -28019.733,E2 -28019.733} C_VEL
LIN {X 0,Y 82.844,Z 602.591,A -85,B 0,C 180,E1 -28026.429,E2 -28026.429} C_VEL
LIN {X 0,Y 88.745,Z 597.571,A -85,B 0,C 180,E1 -28032.309,E2 -28032.309} C_VEL
LIN {X 0,Y 95.455,Z 591.24,A -85,B 0,C 180,E1 -28037.413,E2 -28037.413} C_VEL
LIN {X 0,Y 103.134,Z 582.789,A -85,B 0,C 180,E1 -28042.171,E2 -28042.171} C_VEL
LIN {X 0,Y 110.369,Z 573.482,A -85,B 0,C 180,E1 -28045.872,E2 -28045.872} C_VEL
LIN {X 0,Y 117.191,Z 563.126,A -85,B 0,C 180,E1 -28048.711,E2 -28048.711} C_VEL
LIN {X 0,Y 123.555,Z 551.444,A -85,B 0,C 180,E1 -28050.989,E2 -28050.989} C_VEL
LIN {X 0,Y 128.617,Z 539.765,A -85,B 0,C 180,E1 -28052.614,E2 -28052.614} C_VEL
LIN {X 0,Y 132.557,Z 527.616,A -85,B 0,C 180,E1 -28053.894,E2 -28053.894} C_VEL
LIN {X 0,Y 135.626,Z 514.552,A -85,B 0,C 180,E1 -28054.79,E2 -28054.79} C_VEL
LIN {X 0,Y 137.485,Z 500.75,A -85,B 0,C 180,E1 -28055.39,E2 -28055.39} C_VEL
LIN {X 0,Y 137.965,Z 494.627,A -85,B 0,C 180,E1 -28055.708,E2 -28055.708} C_VEL
LIN {X 0,Y 135.503,Z 488.793,A -85,B 0,C 180,E1 -28058.998,E2 -28058.998} C_VEL
LIN {X 0,Y 132.975,Z 483.441,A -85,B 0,C 180,E1 -28063.051,E2 -28063.051} C_VEL
LIN {X 0,Y 131.212,Z 479.956,A -85,B 0,C 180,E1 -28066.645,E2 -28066.645} C_VEL
LIN {X 0,Y 129.927,Z 477.032,A -85,B 0,C 180,E1 -28070.268,E2 -28070.268} C_VEL
LIN {X 0,Y 128.639,Z 473.047,A -85,B 0,C 180,E1 -28080,E2 -28080} C_VEL
LIN {X 0,Y 130.127,Z 477.526,A -85,B 0,C 180,E1 -28089.913,E2 -28089.913} C_VEL
LIN {X 0,Y 131.935,Z 481.378,A -85,B 0,C 180,E1 -28094.459,E2 -28094.459} C_VEL
LIN {X 0,Y 133.827,Z 485.208,A -85,B 0,C 180,E1 -28097.94,E2 -28097.94} C_VEL
LIN {X 0,Y 135.092,Z 488.191,A -85,B 0,C 180,E1 -28099.963,E2 -28099.963} C_VEL
LIN {X 0,Y 137.081,Z 494.912,A -85,B 0,C 180,E1 -28103.002,E2 -28103.002} C_VEL
LIN {X 0,Y 137.768,Z 497.524,A -85,B 0,C 180,E1 -28103.986,E2 -28103.986} C_VEL
LIN {X 0,Y 135.853,Z 515.055,A -85,B 0,C 180,E1 -28104.696,E2 -28104.696} C_VEL
LIN {X 0,Y 133.089,Z 528.302,A -85,B 0,C 180,E1 -28105.443,E2 -28105.443} C_VEL
LIN {X 0,Y 129.435,Z 540.073,A -85,B 0,C 180,E1 -28106.377,E2 -28106.377} C_VEL
LIN {X 0,Y 124.205,Z 552.717,A -85,B 0,C 180,E1 -28107.859,E2 -28107.859} C_VEL
LIN {X 0,Y 118.337,Z 563.972,A -85,B 0,C 180,E1 -28109.709,E2 -28109.709} C_VEL
LIN {X 0,Y 111.943,Z 574.112,A -85,B 0,C 180,E1 -28112.055,E2 -28112.055} C_VEL
LIN {X 0,Y 105.102,Z 583.257,A -85,B 0,C 180,E1 -28115.003,E2 -28115.003} C_VEL
LIN {X 0,Y 97.382,Z 592.18,A -85,B 0,C 180,E1 -28119.122,E2 -28119.122} C_VEL
LIN {X 0,Y 90.332,Z 599.366,A -85,B 0,C 180,E1 -28123.975,E2 -28123.975} C_VEL
LIN {X 0,Y 83.204,Z 605.925,A -85,B 0,C 180,E1 -28130.692,E2 -28130.692} C_VEL
LIN {X 0,Y 77.959,Z 610.265,A -85,B 0,C 180,E1 -28137.256,E2 -28137.256} C_VEL
LIN {X 0,Y 75.043,Z 612.567,A -85,B 0,C 180,E1 -28142.079,E2 -28142.079} C_VEL
LIN {X 0,Y 72.803,Z 614.437,A -85,B 0,C 180,E1 -28147.286,E2 -28147.286} C_VEL
LIN {X 0,Y 71.184,Z 615.845,A -85,B 0,C 180,E1 -28152.771,E2 -28152.771} C_VEL
LIN {X 0,Y 69.698,Z 617.475,A -85,B 0,C 180,E1 -28164.213,E2 -28164.213} C_VEL
LIN {X 0,Y 69.749,Z 617.696,A -85,B 0,C 180,E1 -28170,E2 -28170} C_VEL
LIN {X 0,Y 69.698,Z 617.457,A -85,B 0,C 180,E1 -28175.787,E2 -28175.787} C_VEL
LIN {X 0,Y 71.181,Z 615.802,A -85,B 0,C 180,E1 -28187.229,E2 -28187.229} C_VEL
LIN {X 0,Y 72.8,Z 614.375,A -85,B 0,C 180,E1 -28192.715,E2 -28192.715} C_VEL
LIN {X 0,Y 76.448,Z 611.404,A -85,B 0,C 180,E1 -28200.372,E2 -28200.372} C_VEL
LIN {X 0,Y 81.304,Z 607.396,A -85,B 0,C 180,E1 -28207.234,E2 -28207.234} C_VEL
LIN {X 0,Y 88.172,Z 601.28,A -85,B 0,C 180,E1 -28214.162,E2 -28214.162} C_VEL
LIN {X 0,Y 94.965,Z 594.532,A -85,B 0,C 180,E1 -28219.336,E2 -28219.336} C_VEL
LIN {X 0,Y 102.483,Z 586.222,A -85,B 0,C 180,E1 -28223.684,E2 -28223.684} C_VEL
LIN {X 0,Y 109.176,Z 577.7,A -85,B 0,C 180,E1 -28226.807,E2 -28226.807} C_VEL
LIN {X 0,Y 116.172,Z 567.178,A -85,B 0,C 180,E1 -28229.548,E2 -28229.548} C_VEL
LIN {X 0,Y 122.71,Z 555.335,A -85,B 0,C 180,E1 -28231.71,E2 -28231.71} C_VEL
LIN {X 0,Y 127.913,Z 543.387,A -85,B 0,C 180,E1 -28233.229,E2 -28233.229} C_VEL
LIN {X 0,Y 132.061,Z 530.947,A -85,B 0,C 180,E1 -28234.337,E2 -28234.337} C_VEL
LIN {X 0,Y 135.127,Z 517.813,A -85,B 0,C 180,E1 -28235.134,E2 -28235.134} C_VEL
LIN {X 0,Y 137.138,Z 502.189,A -85,B 0,C 180,E1 -28235.716,E2 -28235.716} C_VEL
LIN {X 0,Y 137.582,Z 497.576,A -85,B 0,C 180,E1 -28235.879,E2 -28235.879} C_VEL
LIN {X 0,Y 135.696,Z 490.713,A -85,B 0,C 180,E1 -28238.644,E2 -28238.644} C_VEL
LIN {X 0,Y 134.164,Z 486.129,A -85,B 0,C 180,E1 -28241.075,E2 -28241.075} C_VEL
LIN {X 0,Y 132.418,Z 482.677,A -85,B 0,C 180,E1 -28244.019,E2 -28244.019} C_VEL
LIN {X 0,Y 131.121,Z 480.01,A -85,B 0,C 180,E1 -28246.685,E2 -28246.685} C_VEL
LIN {X 0,Y 129.656,Z 476.912,A -85,B 0,C 180,E1 -28250.641,E2 -28250.641} C_VEL
LIN {X 0,Y 128.351,Z 472.629,A -85,B 0,C 180,E1 -28260,E2 -28260} C_VEL
LIN {X 0,Y 128.347,Z 472.997,A -85,B 0,C 180,E1 -28261.765,E2 -28261.765} C_VEL
LIN {X 0,Y 129.348,Z 476.537,A -85,B 0,C 180,E1 -28268.959,E2 -28268.959} C_VEL
LIN {X 0,Y 129.83,Z 477.655,A -85,B 0,C 180,E1 -28270.601,E2 -28270.601} C_VEL
LIN {X 0,Y 130.495,Z 480.568,A -85,B 0,C 180,E1 -28272.843,E2 -28272.843} C_VEL
LIN {X 0,Y 131.122,Z 484.345,A -85,B 0,C 180,E1 -28274.848,E2 -28274.848} C_VEL
LIN {X 0,Y 132.703,Z 492.665,A -85,B 0,C 180,E1 -28278.728,E2 -28278.728} C_VEL
LIN {X 0,Y 133.504,Z 495.068,A -85,B 0,C 180,E1 -28280.109,E2 -28280.109} C_VEL
LIN {X 0,Y 134.704,Z 498.14,A -85,B 0,C 180,E1 -28281.919,E2 -28281.919} C_VEL
LIN {X 0,Y 132.695,Z 513.565,A -85,B 0,C 180,E1 -28282.498,E2 -28282.498} C_VEL
LIN {X 0,Y 129.745,Z 526.263,A -85,B 0,C 180,E1 -28283.265,E2 -28283.265} C_VEL
LIN {X 0,Y 126.197,Z 537.412,A -85,B 0,C 180,E1 -28284.344,E2 -28284.344} C_VEL
LIN {X 0,Y 121.084,Z 549.521,A -85,B 0,C 180,E1 -28285.89,E2 -28285.89} C_VEL
LIN {X 0,Y 115.213,Z 560.526,A -85,B 0,C 180,E1 -28287.813,E2 -28287.813} C_VEL
LIN {X 0,Y 109.449,Z 569.442,A -85,B 0,C 180,E1 -28289.905,E2 -28289.905} C_VEL
LIN {X 0,Y 102.551,Z 578.581,A -85,B 0,C 180,E1 -28292.913,E2 -28292.913} C_VEL
LIN {X 0,Y 94.64,Z 587.464,A -85,B 0,C 180,E1 -28297.034,E2 -28297.034} C_VEL
LIN {X 0,Y 87.238,Z 594.611,A -85,B 0,C 180,E1 -28301.826,E2 -28301.826} C_VEL
LIN {X 0,Y 81.435,Z 599.433,A -85,B 0,C 180,E1 -28306.338,E2 -28306.338} C_VEL
LIN {X 0,Y 75.401,Z 604.107,A -85,B 0,C 180,E1 -28312.711,E2 -28312.711} C_VEL
LIN {X 0,Y 70.331,Z 607.68,A -85,B 0,C 180,E1 -28320.025,E2 -28320.025} C_VEL
LIN {X 0,Y 67.618,Z 609.522,A -85,B 0,C 180,E1 -28325.434,E2 -28325.434} C_VEL
LIN {X 0,Y 65.491,Z 610.903,A -85,B 0,C 180,E1 -28331.22,E2 -28331.22} C_VEL
LIN {X 0,Y 63.107,Z 612.484,A -85,B 0,C 180,E1 -28343.606,E2 -28343.606} C_VEL
LIN {X 0,Y 62.888,Z 612.704,A -85,B 0,C 180,E1 -28350,E2 -28350} C_VEL
LIN {X 0,Y 63.107,Z 612.51,A -85,B 0,C 180,E1 -28356.394,E2 -28356.394} C_VEL
LIN {X 0,Y 65.49,Z 610.961,A -85,B 0,C 180,E1 -28368.78,E2 -28368.78} C_VEL
LIN {X 0,Y 67.61,Z 609.607,A -85,B 0,C 180,E1 -28374.569,E2 -28374.569} C_VEL
LIN {X 0,Y 71.866,Z 606.743,A -85,B 0,C 180,E1 -28382.537,E2 -28382.537} C_VEL
LIN {X 0,Y 77.234,Z 602.857,A -85,B 0,C 180,E1 -28389.565,E2 -28389.565} C_VEL
LIN {X 0,Y 83.642,Z 597.836,A -85,B 0,C 180,E1 -28395.577,E2 -28395.577} C_VEL
LIN {X 0,Y 90.802,Z 591.505,A -85,B 0,C 180,E1 -28400.712,E2 -28400.712} C_VEL
LIN {X 0,Y 98.435,Z 583.61,A -85,B 0,C 180,E1 -28405.167,E2 -28405.167} C_VEL
LIN {X 0,Y 105.169,Z 575.522,A -85,B 0,C 180,E1 -28408.431,E2 -28408.431} C_VEL
LIN {X 0,Y 112.239,Z 565.664,A -85,B 0,C 180,E1 -28411.236,E2 -28411.236} C_VEL
LIN {X 0,Y 118.79,Z 554.55,A -85,B 0,C 180,E1 -28413.486,E2 -28413.486} C_VEL
LIN {X 0,Y 124,Z 543.652,A -85,B 0,C 180,E1 -28415.069,E2 -28415.069} C_VEL
LIN {X 0,Y 128.478,Z 531.599,A -85,B 0,C 180,E1 -28416.382,E2 -28416.382} C_VEL
LIN {X 0,Y 131.837,Z 519.331,A -85,B 0,C 180,E1 -28417.294,E2 -28417.294} C_VEL
LIN {X 0,Y 134.161,Z 505.581,A -85,B 0,C 180,E1 -28417.985,E2 -28417.985} C_VEL
LIN {X 0,Y 134.914,Z 498.278,A -85,B 0,C 180,E1 -28418.274,E2 -28418.274} C_VEL
LIN {X 0,Y 132.606,Z 492.521,A -85,B 0,C 180,E1 -28421.942,E2 -28421.942} C_VEL
LIN {X 0,Y 130.277,Z 487.283,A -85,B 0,C 180,E1 -28426.666,E2 -28426.666} C_VEL
LIN {X 0,Y 128.756,Z 483.852,A -85,B 0,C 180,E1 -28431.169,E2 -28431.169} C_VEL
LIN {X 0,Y 127.758,Z 480.223,A -85,B 0,C 180,E1 -28440,E2 -28440} C_VEL
LIN {X 0,Y 128.973,Z 484.355,A -85,B 0,C 180,E1 -28449.133,E2 -28449.133} C_VEL
LIN {X 0,Y 130.612,Z 488.159,A -85,B 0,C 180,E1 -28453.665,E2 -28453.665} C_VEL
LIN {X 0,Y 132.584,Z 492.469,A -85,B 0,C 180,E1 -28457.534,E2 -28457.534} C_VEL
LIN {X 0,Y 133.967,Z 497.286,A -85,B 0,C 180,E1 -28460.037,E2 -28460.037} C_VEL
LIN {X 0,Y 134.744,Z 500.429,A -85,B 0,C 180,E1 -28461.364,E2 -28461.364} C_VEL
LIN {X 0,Y 132.731,Z 516.676,A -85,B 0,C 180,E1 -28461.999,E2 -28461.999} C_VEL
LIN {X 0,Y 129.878,Z 529.218,A -85,B 0,C 180,E1 -28462.689,E2 -28462.689} C_VEL
LIN {X 0,Y 125.656,Z 541.807,A -85,B 0,C 180,E1 -28463.675,E2 -28463.675} C_VEL
LIN {X 0,Y 120.291,Z 554.039,A -85,B 0,C 180,E1 -28465.1,E2 -28465.1} C_VEL
LIN {X 0,Y 114.241,Z 564.953,A -85,B 0,C 180,E1 -28466.873,E2 -28466.873} C_VEL
LIN {X 0,Y 106.886,Z 575.804,A -85,B 0,C 180,E1 -28469.402,E2 -28469.402} C_VEL
LIN {X 0,Y 99.795,Z 584.626,A -85,B 0,C 180,E1 -28472.32,E2 -28472.32} C_VEL
LIN {X 0,Y 91.737,Z 593.227,A -85,B 0,C 180,E1 -28476.449,E2 -28476.449} C_VEL
LIN {X 0,Y 84.351,Z 600.122,A -85,B 0,C 180,E1 -28481.423,E2 -28481.423} C_VEL
LIN {X 0,Y 77.818,Z 605.658,A -85,B 0,C 180,E1 -28487.365,E2 -28487.365} C_VEL
LIN {X 0,Y 72.071,Z 609.998,A -85,B 0,C 180,E1 -28494.192,E2 -28494.192} C_VEL
LIN {X 0,Y 68.833,Z 612.3,A -85,B 0,C 180,E1 -28499.303,E2 -28499.303} C_VEL
LIN {X 0,Y 66.265,Z 614.168,A -85,B 0,C 180,E1 -28504.898,E2 -28504.898} C_VEL
LIN {X 0,Y 64.416,Z 615.577,A -85,B 0,C 180,E1 -28510.895,E2 -28510.895} C_VEL
LIN {X 0,Y 62.615,Z 617.208,A -85,B 0,C 180,E1 -28523.556,E2 -28523.556} C_VEL
LIN {X 0,Y 62.669,Z 617.429,A -85,B 0,C 180,E1 -28530,E2 -28530} C_VEL
LIN {X 0,Y 62.615,Z 617.188,A -85,B 0,C 180,E1 -28536.444,E2 -28536.444} C_VEL
LIN {X 0,Y 64.413,Z 615.534,A -85,B 0,C 180,E1 -28549.106,E2 -28549.106} C_VEL
LIN {X 0,Y 66.262,Z 614.105,A -85,B 0,C 180,E1 -28555.103,E2 -28555.103} C_VEL
LIN {X 0,Y 70.402,Z 611.135,A -85,B 0,C 180,E1 -28563.301,E2 -28563.301} C_VEL
LIN {X 0,Y 75.757,Z 607.127,A -85,B 0,C 180,E1 -28570.495,E2 -28570.495} C_VEL
LIN {X 0,Y 82.71,Z 601.453,A -85,B 0,C 180,E1 -28577.174,E2 -28577.174} C_VEL
LIN {X 0,Y 90.478,Z 594.261,A -85,B 0,C 180,E1 -28582.766,E2 -28582.766} C_VEL
LIN {X 0,Y 98.442,Z 585.952,A -85,B 0,C 180,E1 -28587.018,E2 -28587.018} C_VEL
LIN {X 0,Y 105.443,Z 577.429,A -85,B 0,C 180,E1 -28590.05,E2 -28590.05} C_VEL
LIN {X 0,Y 112.744,Z 566.907,A -85,B 0,C 180,E1 -28592.656,E2 -28592.656} C_VEL
LIN {X 0,Y 119.513,Z 555.063,A -85,B 0,C 180,E1 -28594.703,E2 -28594.703} C_VEL
LIN {X 0,Y 124.869,Z 543.128,A -85,B 0,C 180,E1 -28596.138,E2 -28596.138} C_VEL
LIN {X 0,Y 129.146,Z 530.671,A -85,B 0,C 180,E1 -28597.176,E2 -28597.176} C_VEL
LIN {X 0,Y 132.133,Z 518.392,A -85,B 0,C 180,E1 -28597.885,E2 -28597.885} C_VEL
LIN {X 0,Y 134.114,Z 504.374,A -85,B 0,C 180,E1 -28598.405,E2 -28598.405} C_VEL
LIN {X 0,Y 134.482,Z 500.206,A -85,B 0,C 180,E1 -28598.6,E2 -28598.6} C_VEL
LIN {X 0,Y 132.731,Z 493.47,A -85,B 0,C 180,E1 -28601.676,E2 -28601.676} C_VEL
LIN {X 0,Y 131.315,Z 489.943,A -85,B 0,C 180,E1 -28604.28,E2 -28604.28} C_VEL
LIN {X 0,Y 129.681,Z 486.458,A -85,B 0,C 180,E1 -28607.878,E2 -28607.878} C_VEL
LIN {X 0,Y 128.542,Z 483.76,A -85,B 0,C 180,E1 -28611.353,E2 -28611.353} C_VEL
LIN {X 0,Y 127.481,Z 479.71,A -85,B 0,C 180,E1 -28620,E2 -28620} C_VEL
LIN {X 0,Y 127.464,Z 480.032,A -85,B 0,C 180,E1 -28621.382,E2 -28621.382} C_VEL
LIN {X 0,Y 128.78,Z 484.323,A -85,B 0,C 180,E1 -28630.054,E2 -28630.054} C_VEL
LIN {X 0,Y 130.398,Z 488.04,A -85,B 0,C 180,E1 -28634.41,E2 -28634.41} C_VEL
LIN {X 0,Y 132.332,Z 492.29,A -85,B 0,C 180,E1 -28638.174,E2 -28638.174} C_VEL
LIN {X 0,Y 133.504,Z 495.068,A -85,B 0,C 180,E1 -28640.109,E2 -28640.109} C_VEL
LIN {X 0,Y 133.782,Z 496.9,A -85,B 0,C 180,E1 -28640.71,E2 -28640.71} C_VEL
LIN {X 0,Y 133.61,Z 499.908,A -85,B 0,C 180,E1 -28640.957,E2 -28640.957} C_VEL
LIN {X 0,Y 132.769,Z 504.388,A -85,B 0,C 180,E1 -28640.707,E2 -28640.707} C_VEL
LIN {X 0,Y 130.417,Z 513.053,A -85,B 0,C 180,E1 -28639.735,E2 -28639.735} C_VEL
LIN {X 0,Y 129.715,Z 516.01,A -85,B 0,C 180,E1 -28639.726,E2 -28639.726} C_VEL
LIN {X 0,Y 126.747,Z 527.803,A -85,B 0,C 180,E1 -28640.441,E2 -28640.441} C_VEL
LIN {X 0,Y 122.607,Z 539.832,A -85,B 0,C 180,E1 -28641.563,E2 -28641.563} C_VEL
LIN {X 0,Y 117.407,Z 551.35,A -85,B 0,C 180,E1 -28643.026,E2 -28643.026} C_VEL
LIN {X 0,Y 110.575,Z 563.143,A -85,B 0,C 180,E1 -28645.083,E2 -28645.083} C_VEL
LIN {X 0,Y 103.155,Z 573.603,A -85,B 0,C 180,E1 -28647.665,E2 -28647.665} C_VEL
LIN {X 0,Y 94.993,Z 583.163,A -85,B 0,C 180,E1 -28651.191,E2 -28651.191} C_VEL
LIN {X 0,Y 86.55,Z 591.502,A -85,B 0,C 180,E1 -28655.709,E2 -28655.709} C_VEL
LIN {X 0,Y 78.907,Z 597.896,A -85,B 0,C 180,E1 -28660.795,E2 -28660.795} C_VEL
LIN {X 0,Y 71.941,Z 602.966,A -85,B 0,C 180,E1 -28666.857,E2 -28666.857} C_VEL
LIN {X 0,Y 66.026,Z 606.893,A -85,B 0,C 180,E1 -28674.167,E2 -28674.167} C_VEL
LIN {X 0,Y 61.24,Z 609.79,A -85,B 0,C 180,E1 -28682.675,E2 -28682.675} C_VEL
LIN {X 0,Y 57.089,Z 612.151,A -85,B 0,C 180,E1 -28695.747,E2 -28695.747} C_VEL
LIN {X 0,Y 56.083,Z 612.75,A -85,B 0,C 180,E1 -28702.801,E2 -28702.801} C_VEL
LIN {X 0,Y 55.81,Z 612.971,A -85,B 0,C 180,E1 -28710,E2 -28710} C_VEL
LIN {X 0,Y 56.083,Z 612.776,A -85,B 0,C 180,E1 -28717.199,E2 -28717.199} C_VEL
LIN {X 0,Y 58.807,Z 611.228,A -85,B 0,C 180,E1 -28731.009,E2 -28731.009} C_VEL
LIN {X 0,Y 61.232,Z 609.873,A -85,B 0,C 180,E1 -28737.329,E2 -28737.329} C_VEL
LIN {X 0,Y 65.984,Z 607.01,A -85,B 0,C 180,E1 -28745.859,E2 -28745.859} C_VEL
LIN {X 0,Y 71.893,Z 603.124,A -85,B 0,C 180,E1 -28753.179,E2 -28753.179} C_VEL
LIN {X 0,Y 78.847,Z 598.101,A -85,B 0,C 180,E1 -28759.256,E2 -28759.256} C_VEL
LIN {X 0,Y 86.484,Z 591.77,A -85,B 0,C 180,E1 -28764.352,E2 -28764.352} C_VEL
LIN {X 0,Y 94.029,Z 584.435,A -85,B 0,C 180,E1 -28768.453,E2 -28768.453} C_VEL
LIN {X 0,Y 101.633,Z 575.786,A -85,B 0,C 180,E1 -28771.842,E2 -28771.842} C_VEL
LIN {X 0,Y 109.003,Z 565.928,A -85,B 0,C 180,E1 -28774.506,E2 -28774.506} C_VEL
LIN {X 0,Y 115.797,Z 554.813,A -85,B 0,C 180,E1 -28776.629,E2 -28776.629} C_VEL
LIN {X 0,Y 121.18,Z 543.913,A -85,B 0,C 180,E1 -28778.112,E2 -28778.112} C_VEL
LIN {X 0,Y 125.928,Z 531.507,A -85,B 0,C 180,E1 -28779.37,E2 -28779.37} C_VEL
LIN {X 0,Y 129.44,Z 518.735,A -85,B 0,C 180,E1 -28780.249,E2 -28780.249} C_VEL
LIN {X 0,Y 131.777,Z 504.981,A -85,B 0,C 180,E1 -28780.873,E2 -28780.873} C_VEL
LIN {X 0,Y 132.077,Z 501.947,A -85,B 0,C 180,E1 -28781.038,E2 -28781.038} C_VEL
LIN {X 0,Y 130.03,Z 496.565,A -85,B 0,C 180,E1 -28785.018,E2 -28785.018} C_VEL
LIN {X 0,Y 128.474,Z 492.903,A -85,B 0,C 180,E1 -28788.962,E2 -28788.962} C_VEL
LIN {X 0,Y 127.621,Z 490.639,A -85,B 0,C 180,E1 -28792.087,E2 -28792.087} C_VEL
LIN {X 0,Y 126.874,Z 487.425,A -85,B 0,C 180,E1 -28800,E2 -28800} C_VEL
LIN {X 0,Y 127.895,Z 491.282,A -85,B 0,C 180,E1 -28808.529,E2 -28808.529} C_VEL
LIN {X 0,Y 129.238,Z 494.749,A -85,B 0,C 180,E1 -28812.663,E2 -28812.663} C_VEL
LIN {X 0,Y 130.877,Z 498.752,A -85,B 0,C 180,E1 -28816.266,E2 -28816.266} C_VEL
LIN {X 0,Y 131.948,Z 503.289,A -85,B 0,C 180,E1 -28818.536,E2 -28818.536} C_VEL
LIN {X 0,Y 130.426,Z 515.318,A -85,B 0,C 180,E1 -28819.055,E2 -28819.055} C_VEL
LIN {X 0,Y 127.4,Z 528.645,A -85,B 0,C 180,E1 -28819.721,E2 -28819.721} C_VEL
LIN {X 0,Y 122.924,Z 541.686,A -85,B 0,C 180,E1 -28820.66,E2 -28820.66} C_VEL
LIN {X 0,Y 117.459,Z 553.777,A -85,B 0,C 180,E1 -28821.967,E2 -28821.967} C_VEL
LIN {X 0,Y 111.214,Z 564.69,A -85,B 0,C 180,E1 -28823.611,E2 -28823.611} C_VEL
LIN {X 0,Y 103.585,Z 575.54,A -85,B 0,C 180,E1 -28825.979,E2 -28825.979} C_VEL
LIN {X 0,Y 96.187,Z 584.361,A -85,B 0,C 180,E1 -28828.745,E2 -28828.745} C_VEL
LIN {X 0,Y 89.083,Z 591.648,A -85,B 0,C 180,E1 -28831.996,E2 -28831.996} C_VEL
LIN {X 0,Y 81.074,Z 598.832,A -85,B 0,C 180,E1 -28836.695,E2 -28836.695} C_VEL
LIN {X 0,Y 74.968,Z 603.692,A -85,B 0,C 180,E1 -28841.414,E2 -28841.414} C_VEL
LIN {X 0,Y 68.368,Z 608.418,A -85,B 0,C 180,E1 -28848.074,E2 -28848.074} C_VEL
LIN {X 0,Y 62.821,Z 612.033,A -85,B 0,C 180,E1 -28855.989,E2 -28855.989} C_VEL
LIN {X 0,Y 59.87,Z 613.9,A -85,B 0,C 180,E1 -28861.995,E2 -28861.995} C_VEL
LIN {X 0,Y 57.706,Z 615.308,A -85,B 0,C 180,E1 -28868.57,E2 -28868.57} C_VEL
LIN {X 0,Y 56.26,Z 616.319,A -85,B 0,C 180,E1 -28875.532,E2 -28875.532} C_VEL
LIN {X 0,Y 55.557,Z 616.94,A -85,B 0,C 180,E1 -28882.733,E2 -28882.733} C_VEL
LIN {X 0,Y 55.578,Z 617.162,A -85,B 0,C 180,E1 -28890,E2 -28890} C_VEL
LIN {X 0,Y 55.557,Z 616.921,A -85,B 0,C 180,E1 -28897.267,E2 -28897.267} C_VEL
LIN {X 0,Y 56.259,Z 616.287,A -85,B 0,C 180,E1 -28904.468,E2 -28904.468} C_VEL
LIN {X 0,Y 57.703,Z 615.264,A -85,B 0,C 180,E1 -28911.431,E2 -28911.431} C_VEL
LIN {X 0,Y 59.867,Z 613.836,A -85,B 0,C 180,E1 -28918.006,E2 -28918.006} C_VEL
LIN {X 0,Y 64.551,Z 610.865,A -85,B 0,C 180,E1 -28926.784,E2 -28926.784} C_VEL
LIN {X 0,Y 70.496,Z 606.858,A -85,B 0,C 180,E1 -28934.254,E2 -28934.254} C_VEL
LIN {X 0,Y 77.458,Z 601.658,A -85,B 0,C 180,E1 -28940.571,E2 -28940.571} C_VEL
LIN {X 0,Y 85.012,Z 595.23,A -85,B 0,C 180,E1 -28945.76,E2 -28945.76} C_VEL
LIN {X 0,Y 93.316,Z 587.174,A -85,B 0,C 180,E1 -28950.007,E2 -28950.007} C_VEL
LIN {X 0,Y 100.599,Z 578.968,A -85,B 0,C 180,E1 -28952.963,E2 -28952.963} C_VEL
LIN {X 0,Y 108.127,Z 568.965,A -85,B 0,C 180,E1 -28955.498,E2 -28955.498} C_VEL
LIN {X 0,Y 115.087,Z 557.653,A -85,B 0,C 180,E1 -28957.46,E2 -28957.46} C_VEL
LIN {X 0,Y 120.586,Z 546.569,A -85,B 0,C 180,E1 -28958.827,E2 -28958.827} C_VEL
LIN {X 0,Y 125.061,Z 535.116,A -85,B 0,C 180,E1 -28959.823,E2 -28959.823} C_VEL
LIN {X 0,Y 128.664,Z 522.546,A -85,B 0,C 180,E1 -28960.587,E2 -28960.587} C_VEL
LIN {X 0,Y 131.069,Z 509.143,A -85,B 0,C 180,E1 -28961.13,E2 -28961.13} C_VEL
LIN {X 0,Y 131.73,Z 503.283,A -85,B 0,C 180,E1 -28961.331,E2 -28961.331} C_VEL
LIN {X 0,Y 130.568,Z 498.354,A -85,B 0,C 180,E1 -28963.786,E2 -28963.786} C_VEL
LIN {X 0,Y 128.644,Z 493.542,A -85,B 0,C 180,E1 -28968.178,E2 -28968.178} C_VEL
LIN {X 0,Y 127.346,Z 490.44,A -85,B 0,C 180,E1 -28972.469,E2 -28972.469} C_VEL
LIN {X 0,Y 126.606,Z 486.839,A -85,B 0,C 180,E1 -28980,E2 -28980} C_VEL
LIN {X 0,Y 126.571,Z 487.757,A -85,B 0,C 180,E1 -28982.308,E2 -28982.308} C_VEL
LIN {X 0,Y 127.654,Z 491.152,A -85,B 0,C 180,E1 -28989.307,E2 -28989.307} C_VEL
LIN {X 0,Y 129.083,Z 494.819,A -85,B 0,C 180,E1 -28993.58,E2 -28993.58} C_VEL
LIN {X 0,Y 130.77,Z 498.943,A -85,B 0,C 180,E1 -28997.193,E2 -28997.193} C_VEL
LIN {X 0,Y 131.845,Z 501.841,A -85,B 0,C 180,E1 -28999.153,E2 -28999.153} C_VEL
LIN {X 0,Y 129.986,Z 514.711,A -85,B 0,C 180,E1 -28999.652,E2 -28999.652} C_VEL
LIN {X 0,Y 129.715,Z 516.01,A -85,B 0,C 180,E1 -28999.726,E2 -28999.726} C_VEL
LIN {X 0,Y 127.538,Z 523.59,A -85,B 0,C 180,E1 -28999.642,E2 -28999.642} C_VEL
LIN {X 0,Y 124.601,Z 530.898,A -85,B 0,C 180,E1 -28999.074,E2 -28999.074} C_VEL
LIN {X 0,Y 120.436,Z 539.891,A -85,B 0,C 180,E1 -28998.639,E2 -28998.639} C_VEL
LIN {X 0,Y 117.965,Z 545.162,A -85,B 0,C 180,E1 -28998.934,E2 -28998.934} C_VEL
LIN {X 0,Y 112.449,Z 555.892,A -85,B 0,C 180,E1 -29000.369,E2 -29000.369} C_VEL
LIN {X 0,Y 105.417,Z 566.801,A -85,B 0,C 180,E1 -29002.331,E2 -29002.331} C_VEL
LIN {X 0,Y 98.549,Z 575.669,A -85,B 0,C 180,E1 -29004.6,E2 -29004.6} C_VEL
LIN {X 0,Y 91.145,Z 583.816,A -85,B 0,C 180,E1 -29007.558,E2 -29007.558} C_VEL
LIN {X 0,Y 82.609,Z 591.771,A -85,B 0,C 180,E1 -29011.708,E2 -29011.708} C_VEL
LIN {X 0,Y 74.473,Z 598.164,A -85,B 0,C 180,E1 -29016.666,E2 -29016.666} C_VEL
LIN {X 0,Y 66.931,Z 603.234,A -85,B 0,C 180,E1 -29022.692,E2 -29022.692} C_VEL
LIN {X 0,Y 60.409,Z 607.161,A -85,B 0,C 180,E1 -29030.219,E2 -29030.219} C_VEL
LIN {X 0,Y 55.043,Z 610.057,A -85,B 0,C 180,E1 -29039.289,E2 -29039.289} C_VEL
LIN {X 0,Y 50.247,Z 612.418,A -85,B 0,C 180,E1 -29053.756,E2 -29053.756} C_VEL
LIN {X 0,Y 49.061,Z 613.017,A -85,B 0,C 180,E1 -29061.764,E2 -29061.764} C_VEL
LIN {X 0,Y 48.73,Z 613.237,A -85,B 0,C 180,E1 -29070,E2 -29070} C_VEL
LIN {X 0,Y 49.061,Z 613.042,A -85,B 0,C 180,E1 -29078.236,E2 -29078.236} C_VEL
LIN {X 0,Y 52.248,Z 611.495,A -85,B 0,C 180,E1 -29093.799,E2 -29093.799} C_VEL
LIN {X 0,Y 55.01,Z 610.14,A -85,B 0,C 180,E1 -29100.732,E2 -29100.732} C_VEL
LIN {X 0,Y 60.375,Z 607.276,A -85,B 0,C 180,E1 -29109.808,E2 -29109.808} C_VEL
LIN {X 0,Y 66.885,Z 603.39,A -85,B 0,C 180,E1 -29117.351,E2 -29117.351} C_VEL
LIN {X 0,Y 74.418,Z 598.366,A -85,B 0,C 180,E1 -29123.39,E2 -29123.39} C_VEL
LIN {X 0,Y 82.552,Z 592.035,A -85,B 0,C 180,E1 -29128.356,E2 -29128.356} C_VEL
LIN {X 0,Y 90.861,Z 584.348,A -85,B 0,C 180,E1 -29132.442,E2 -29132.442} C_VEL
LIN {X 0,Y 98.488,Z 576.05,A -85,B 0,C 180,E1 -29135.478,E2 -29135.478} C_VEL
LIN {X 0,Y 106.141,Z 566.191,A -85,B 0,C 180,E1 -29137.968,E2 -29137.968} C_VEL
LIN {X 0,Y 113.176,Z 555.075,A -85,B 0,C 180,E1 -29139.92,E2 -29139.92} C_VEL
LIN {X 0,Y 119.444,Z 542.62,A -85,B 0,C 180,E1 -29141.422,E2 -29141.422} C_VEL
LIN {X 0,Y 123.889,Z 530.955,A -85,B 0,C 180,E1 -29142.509,E2 -29142.509} C_VEL
LIN {X 0,Y 127.5,Z 517.689,A -85,B 0,C 180,E1 -29143.325,E2 -29143.325} C_VEL
LIN {X 0,Y 129.503,Z 505.972,A -85,B 0,C 180,E1 -29143.852,E2 -29143.852} C_VEL
LIN {X 0,Y 128.102,Z 501.888,A -85,B 0,C 180,E1 -29147.323,E2 -29147.323} C_VEL
LIN {X 0,Y 126.902,Z 498.59,A -85,B 0,C 180,E1 -29151.24,E2 -29151.24} C_VEL
LIN {X 0,Y 126.484,Z 497.296,A -85,B 0,C 180,E1 -29153.219,E2 -29153.219} C_VEL
LIN {X 0,Y 125.992,Z 494.612,A -85,B 0,C 180,E1 -29160,E2 -29160} C_VEL
LIN {X 0,Y 126.752,Z 497.985,A -85,B 0,C 180,E1 -29167.567,E2 -29167.567} C_VEL
LIN {X 0,Y 127.888,Z 501.29,A -85,B 0,C 180,E1 -29171.591,E2 -29171.591} C_VEL
LIN {X 0,Y 129.152,Z 504.805,A -85,B 0,C 180,E1 -29174.778,E2 -29174.778} C_VEL
LIN {X 0,Y 129.52,Z 506.615,A -85,B 0,C 180,E1 -29175.742,E2 -29175.742} C_VEL
LIN {X 0,Y 127.288,Z 520.023,A -85,B 0,C 180,E1 -29176.252,E2 -29176.252} C_VEL
LIN {X 0,Y 123.757,Z 532.956,A -85,B 0,C 180,E1 -29176.931,E2 -29176.931} C_VEL
LIN {X 0,Y 118.962,Z 545.303,A -85,B 0,C 180,E1 -29177.828,E2 -29177.828} C_VEL
LIN {X 0,Y 112.571,Z 557.883,A -85,B 0,C 180,E1 -29179.221,E2 -29179.221} C_VEL
LIN {X 0,Y 105.383,Z 569.073,A -85,B 0,C 180,E1 -29180.991,E2 -29180.991} C_VEL
LIN {X 0,Y 97.555,Z 579.008,A -85,B 0,C 180,E1 -29183.291,E2 -29183.291} C_VEL
LIN {X 0,Y 88.46,Z 588.648,A -85,B 0,C 180,E1 -29186.649,E2 -29186.649} C_VEL
LIN {X 0,Y 79.781,Z 596.325,A -85,B 0,C 180,E1 -29190.811,E2 -29190.811} C_VEL
LIN {X 0,Y 70.43,Z 603.424,A -85,B 0,C 180,E1 -29197.035,E2 -29197.035} C_VEL
LIN {X 0,Y 63.238,Z 608.15,A -85,B 0,C 180,E1 -29203.75,E2 -29203.75} C_VEL
LIN {X 0,Y 57.063,Z 611.766,A -85,B 0,C 180,E1 -29211.99,E2 -29211.99} C_VEL
LIN {X 0,Y 53.668,Z 613.632,A -85,B 0,C 180,E1 -29218.412,E2 -29218.412} C_VEL
LIN {X 0,Y 49.38,Z 616.051,A -85,B 0,C 180,E1 -29233.463,E2 -29233.463} C_VEL
LIN {X 0,Y 48.506,Z 616.673,A -85,B 0,C 180,E1 -29241.669,E2 -29241.669} C_VEL
LIN {X 0,Y 48.476,Z 616.895,A -85,B 0,C 180,E1 -29250,E2 -29250} C_VEL
LIN {X 0,Y 48.506,Z 616.653,A -85,B 0,C 180,E1 -29258.331,E2 -29258.331} C_VEL
LIN {X 0,Y 49.379,Z 616.018,A -85,B 0,C 180,E1 -29266.538,E2 -29266.538} C_VEL
LIN {X 0,Y 51.117,Z 614.995,A -85,B 0,C 180,E1 -29274.359,E2 -29274.359} C_VEL
LIN {X 0,Y 53.665,Z 613.566,A -85,B 0,C 180,E1 -29281.589,E2 -29281.589} C_VEL
LIN {X 0,Y 58.991,Z 610.596,A -85,B 0,C 180,E1 -29290.938,E2 -29290.938} C_VEL
LIN {X 0,Y 65.588,Z 606.589,A -85,B 0,C 180,E1 -29298.595,E2 -29298.595} C_VEL
LIN {X 0,Y 73.356,Z 601.222,A -85,B 0,C 180,E1 -29305.051,E2 -29305.051} C_VEL
LIN {X 0,Y 82.634,Z 593.721,A -85,B 0,C 180,E1 -29310.661,E2 -29310.661} C_VEL
LIN {X 0,Y 91.469,Z 585.411,A -85,B 0,C 180,E1 -29314.527,E2 -29314.527} C_VEL
LIN {X 0,Y 99.103,Z 576.887,A -85,B 0,C 180,E1 -29317.203,E2 -29317.203} C_VEL
LIN {X 0,Y 106.976,Z 566.367,A -85,B 0,C 180,E1 -29319.417,E2 -29319.417} C_VEL
LIN {X 0,Y 113.365,Z 555.954,A -85,B 0,C 180,E1 -29320.978,E2 -29320.978} C_VEL
LIN {X 0,Y 118.928,Z 544.747,A -85,B 0,C 180,E1 -29322.168,E2 -29322.168} C_VEL
LIN {X 0,Y 123.47,Z 532.845,A -85,B 0,C 180,E1 -29323.064,E2 -29323.064} C_VEL
LIN {X 0,Y 127.155,Z 519.268,A -85,B 0,C 180,E1 -29323.74,E2 -29323.74} C_VEL
LIN {X 0,Y 129.245,Z 506.423,A -85,B 0,C 180,E1 -29324.224,E2 -29324.224} C_VEL
LIN {X 0,Y 128.714,Z 504.032,A -85,B 0,C 180,E1 -29325.575,E2 -29325.575} C_VEL
LIN {X 0,Y 127.128,Z 499.708,A -85,B 0,C 180,E1 -29329.851,E2 -29329.851} C_VEL
LIN {X 0,Y 126.285,Z 497.282,A -85,B 0,C 180,E1 -29333.208,E2 -29333.208} C_VEL
LIN {X 0,Y 125.716,Z 494.088,A -85,B 0,C 180,E1 -29340,E2 -29340} C_VEL
LIN {X 0,Y 125.714,Z 495.423,A -85,B 0,C 180,E1 -29343.205,E2 -29343.205} C_VEL
LIN {X 0,Y 126.512,Z 497.869,A -85,B 0,C 180,E1 -29348.385,E2 -29348.385} C_VEL
LIN {X 0,Y 127.717,Z 501.371,A -85,B 0,C 180,E1 -29352.514,E2 -29352.514} C_VEL
LIN {X 0,Y 129.117,Z 505.353,A -85,B 0,C 180,E1 -29355.995,E2 -29355.995} C_VEL
LIN {X 0,Y 129.234,Z 505.745,A -85,B 0,C 180,E1 -29356.271,E2 -29356.271} C_VEL
LIN {X 0,Y 126.893,Z 519.08,A -85,B 0,C 180,E1 -29356.871,E2 -29356.871} C_VEL
LIN {X 0,Y 123.619,Z 530.83,A -85,B 0,C 180,E1 -29357.602,E2 -29357.602} C_VEL
LIN {X 0,Y 119.415,Z 541.958,A -85,B 0,C 180,E1 -29358.599,E2 -29358.599} C_VEL
LIN {X 0,Y 117.965,Z 545.162,A -85,B 0,C 180,E1 -29358.934,E2 -29358.934} C_VEL
LIN {X 0,Y 115.275,Z 550.394,A -85,B 0,C 180,E1 -29359.261,E2 -29359.261} C_VEL
LIN {X 0,Y 109.779,Z 558.664,A -85,B 0,C 180,E1 -29359.029,E2 -29359.029} C_VEL
LIN {X 0,Y 103.648,Z 566.47,A -85,B 0,C 180,E1 -29358.907,E2 -29358.907} C_VEL
LIN {X 0,Y 99.963,Z 570.97,A -85,B 0,C 180,E1 -29359.501,E2 -29359.501} C_VEL
LIN {X 0,Y 92.711,Z 579.391,A -85,B 0,C 180,E1 -29361.783,E2 -29361.783} C_VEL
LIN {X 0,Y 83.56,Z 588.272,A -85,B 0,C 180,E1 -29365.294,E2 -29365.294} C_VEL
LIN {X 0,Y 74.739,Z 595.418,A -85,B 0,C 180,E1 -29369.566,E2 -29369.566} C_VEL
LIN {X 0,Y 67.673,Z 600.237,A -85,B 0,C 180,E1 -29373.819,E2 -29373.819} C_VEL
LIN {X 0,Y 59.846,Z 604.913,A -85,B 0,C 180,E1 -29380.243,E2 -29380.243} C_VEL
LIN {X 0,Y 52.969,Z 608.484,A -85,B 0,C 180,E1 -29388.441,E2 -29388.441} C_VEL
LIN {X 0,Y 49.064,Z 610.325,A -85,B 0,C 180,E1 -29395.044,E2 -29395.044} C_VEL
LIN {X 0,Y 45.859,Z 611.705,A -85,B 0,C 180,E1 -29402.629,E2 -29402.629} C_VEL
LIN {X 0,Y 42.05,Z 613.284,A -85,B 0,C 180,E1 -29420.379,E2 -29420.379} C_VEL
LIN {X 0,Y 41.637,Z 613.504,A -85,B 0,C 180,E1 -29430,E2 -29430} C_VEL
LIN {X 0,Y 42.05,Z 613.309,A -85,B 0,C 180,E1 -29439.621,E2 -29439.621} C_VEL
LIN {X 0,Y 45.856,Z 611.761,A -85,B 0,C 180,E1 -29457.373,E2 -29457.373} C_VEL
LIN {X 0,Y 49.037,Z 610.407,A -85,B 0,C 180,E1 -29464.978,E2 -29464.978} C_VEL
LIN {X 0,Y 55.113,Z 607.542,A -85,B 0,C 180,E1 -29474.534,E2 -29474.534} C_VEL
LIN {X 0,Y 62.287,Z 603.657,A -85,B 0,C 180,E1 -29482.167,E2 -29482.167} C_VEL
LIN {X 0,Y 70.417,Z 598.631,A -85,B 0,C 180,E1 -29488.03,E2 -29488.03} C_VEL
LIN {X 0,Y 79.061,Z 592.3,A -85,B 0,C 180,E1 -29492.737,E2 -29492.737} C_VEL
LIN {X 0,Y 88.033,Z 584.39,A -85,B 0,C 180,E1 -29496.64,E2 -29496.64} C_VEL
LIN {X 0,Y 95.761,Z 576.314,A -85,B 0,C 180,E1 -29499.344,E2 -29499.344} C_VEL
LIN {X 0,Y 103.693,Z 566.454,A -85,B 0,C 180,E1 -29501.596,E2 -29501.596} C_VEL
LIN {X 0,Y 110.939,Z 555.337,A -85,B 0,C 180,E1 -29503.365,E2 -29503.365} C_VEL
LIN {X 0,Y 117.326,Z 543.001,A -85,B 0,C 180,E1 -29504.686,E2 -29504.686} C_VEL
LIN {X 0,Y 121.948,Z 531.214,A -85,B 0,C 180,E1 -29505.684,E2 -29505.684} C_VEL
LIN {X 0,Y 125.471,Z 518.769,A -85,B 0,C 180,E1 -29506.374,E2 -29506.374} C_VEL
LIN {X 0,Y 127.171,Z 510.201,A -85,B 0,C 180,E1 -29506.725,E2 -29506.725} C_VEL
LIN {X 0,Y 126.058,Z 506.287,A -85,B 0,C 180,E1 -29510.776,E2 -29510.776} C_VEL
LIN {X 0,Y 125.459,Z 504.147,A -85,B 0,C 180,E1 -29513.971,E2 -29513.971} C_VEL
LIN {X 0,Y 125.111,Z 501.783,A -85,B 0,C 180,E1 -29520,E2 -29520} C_VEL
LIN {X 0,Y 125.685,Z 504.876,A -85,B 0,C 180,E1 -29526.824,E2 -29526.824} C_VEL
LIN {X 0,Y 126.51,Z 507.77,A -85,B 0,C 180,E1 -29530.401,E2 -29530.401} C_VEL
LIN {X 0,Y 127.252,Z 510.167,A -85,B 0,C 180,E1 -29532.763,E2 -29532.763} C_VEL
LIN {X 0,Y 124.856,Z 522.527,A -85,B 0,C 180,E1 -29533.242,E2 -29533.242} C_VEL
LIN {X 0,Y 120.896,Z 535.45,A -85,B 0,C 180,E1 -29533.883,E2 -29533.883} C_VEL
LIN {X 0,Y 116.219,Z 546.66,A -85,B 0,C 180,E1 -29534.64,E2 -29534.64} C_VEL
LIN {X 0,Y 110.437,Z 557.62,A -85,B 0,C 180,E1 -29535.741,E2 -29535.741} C_VEL
LIN {X 0,Y 103.049,Z 568.809,A -85,B 0,C 180,E1 -29537.296,E2 -29537.296} C_VEL
LIN {X 0,Y 94.965,Z 578.743,A -85,B 0,C 180,E1 -29539.342,E2 -29539.342} C_VEL
LIN {X 0,Y 85.507,Z 588.383,A -85,B 0,C 180,E1 -29542.386,E2 -29542.386} C_VEL
LIN {X 0,Y 76.376,Z 596.059,A -85,B 0,C 180,E1 -29546.214,E2 -29546.214} C_VEL
LIN {X 0,Y 66.369,Z 603.156,A -85,B 0,C 180,E1 -29552.1,E2 -29552.1} C_VEL
LIN {X 0,Y 58.536,Z 607.883,A -85,B 0,C 180,E1 -29558.703,E2 -29558.703} C_VEL
LIN {X 0,Y 51.622,Z 611.498,A -85,B 0,C 180,E1 -29567.102,E2 -29567.102} C_VEL
LIN {X 0,Y 47.733,Z 613.364,A -85,B 0,C 180,E1 -29573.919,E2 -29573.919} C_VEL
LIN {X 0,Y 42.595,Z 615.783,A -85,B 0,C 180,E1 -29590.732,E2 -29590.732} C_VEL
LIN {X 0,Y 41.471,Z 616.405,A -85,B 0,C 180,E1 -29600.243,E2 -29600.243} C_VEL
LIN {X 0,Y 41.392,Z 616.629,A -85,B 0,C 180,E1 -29610,E2 -29610} C_VEL
LIN {X 0,Y 41.471,Z 616.384,A -85,B 0,C 180,E1 -29619.757,E2 -29619.757} C_VEL
LIN {X 0,Y 42.593,Z 615.75,A -85,B 0,C 180,E1 -29629.269,E2 -29629.269} C_VEL
LIN {X 0,Y 44.712,Z 614.726,A -85,B 0,C 180,E1 -29638.134,E2 -29638.134} C_VEL
LIN {X 0,Y 47.73,Z 613.297,A -85,B 0,C 180,E1 -29646.083,E2 -29646.083} C_VEL
LIN {X 0,Y 53.804,Z 610.327,A -85,B 0,C 180,E1 -29655.923,E2 -29655.923} C_VEL
LIN {X 0,Y 61.113,Z 606.32,A -85,B 0,C 180,E1 -29663.609,E2 -29663.609} C_VEL
LIN {X 0,Y 69.981,Z 600.618,A -85,B 0,C 180,E1 -29670.164,E2 -29670.164} C_VEL
LIN {X 0,Y 79.387,Z 593.451,A -85,B 0,C 180,E1 -29675.147,E2 -29675.147} C_VEL
LIN {X 0,Y 88.641,Z 585.141,A -85,B 0,C 180,E1 -29678.683,E2 -29678.683} C_VEL
LIN {X 0,Y 96.57,Z 576.616,A -85,B 0,C 180,E1 -29681.097,E2 -29681.097} C_VEL
LIN {X 0,Y 104.688,Z 566.095,A -85,B 0,C 180,E1 -29683.061,E2 -29683.061} C_VEL
LIN {X 0,Y 111.25,Z 555.682,A -85,B 0,C 180,E1 -29684.443,E2 -29684.443} C_VEL
LIN {X 0,Y 116.892,Z 544.598,A -85,B 0,C 180,E1 -29685.471,E2 -29685.471} C_VEL
LIN {X 0,Y 121.596,Z 532.57,A -85,B 0,C 180,E1 -29686.256,E2 -29686.256} C_VEL
LIN {X 0,Y 125.255,Z 519.431,A -85,B 0,C 180,E1 -29686.836,E2 -29686.836} C_VEL
LIN {X 0,Y 126.979,Z 509.909,A -85,B 0,C 180,E1 -29687.209,E2 -29687.209} C_VEL
LIN {X 0,Y 125.822,Z 506.125,A -85,B 0,C 180,E1 -29691.164,E2 -29691.164} C_VEL
LIN {X 0,Y 125.246,Z 504.116,A -85,B 0,C 180,E1 -29693.961,E2 -29693.961} C_VEL
LIN {X 0,Y 124.829,Z 501.309,A -85,B 0,C 180,E1 -29700,E2 -29700} C_VEL
LIN {X 0,Y 124.994,Z 503.457,A -85,B 0,C 180,E1 -29705.04,E2 -29705.04} C_VEL
LIN {X 0,Y 125.469,Z 504.895,A -85,B 0,C 180,E1 -29707.848,E2 -29707.848} C_VEL
LIN {X 0,Y 126.4,Z 508.199,A -85,B 0,C 180,E1 -29711.73,E2 -29711.73} C_VEL
LIN {X 0,Y 126.891,Z 509.935,A -85,B 0,C 180,E1 -29713.354,E2 -29713.354} C_VEL
LIN {X 0,Y 124.044,Z 523.105,A -85,B 0,C 180,E1 -29713.915,E2 -29713.915} C_VEL
LIN {X 0,Y 119.801,Z 536.311,A -85,B 0,C 180,E1 -29714.828,E2 -29714.828} C_VEL
LIN {X 0,Y 115.049,Z 547.181,A -85,B 0,C 180,E1 -29715.826,E2 -29715.826} C_VEL
LIN {X 0,Y 108.571,Z 558.778,A -85,B 0,C 180,E1 -29717.298,E2 -29717.298} C_VEL
LIN {X 0,Y 101.335,Z 569.201,A -85,B 0,C 180,E1 -29719.103,E2 -29719.103} C_VEL
LIN {X 0,Y 99.963,Z 570.97,A -85,B 0,C 180,E1 -29719.501,E2 -29719.501} C_VEL
LIN {X 0,Y 96.121,Z 575.366,A -85,B 0,C 180,E1 -29720.221,E2 -29720.221} C_VEL
LIN {X 0,Y 88.905,Z 582.167,A -85,B 0,C 180,E1 -29720.602,E2 -29720.602} C_VEL
LIN {X 0,Y 81.253,Z 588.355,A -85,B 0,C 180,E1 -29721.161,E2 -29721.161} C_VEL
LIN {X 0,Y 76.775,Z 591.79,A -85,B 0,C 180,E1 -29722.318,E2 -29722.318} C_VEL
LIN {X 0,Y 66.979,Z 598.701,A -85,B 0,C 180,E1 -29726.89,E2 -29726.89} C_VEL
LIN {X 0,Y 58.237,Z 603.772,A -85,B 0,C 180,E1 -29732.356,E2 -29732.356} C_VEL
LIN {X 0,Y 50.315,Z 607.698,A -85,B 0,C 180,E1 -29739.806,E2 -29739.806} C_VEL
LIN {X 0,Y 43.435,Z 610.593,A -85,B 0,C 180,E1 -29749.669,E2 -29749.669} C_VEL
LIN {X 0,Y 39.686,Z 611.972,A -85,B 0,C 180,E1 -29757.91,E2 -29757.91} C_VEL
LIN {X 0,Y 35.09,Z 613.551,A -85,B 0,C 180,E1 -29778.447,E2 -29778.447} C_VEL
LIN {X 0,Y 34.564,Z 613.77,A -85,B 0,C 180,E1 -29790,E2 -29790} C_VEL
LIN {X 0,Y 35.09,Z 613.575,A -85,B 0,C 180,E1 -29801.553,E2 -29801.553} C_VEL
LIN {X 0,Y 39.682,Z 612.028,A -85,B 0,C 180,E1 -29822.094,E2 -29822.094} C_VEL
LIN {X 0,Y 43.413,Z 610.673,A -85,B 0,C 180,E1 -29830.356,E2 -29830.356} C_VEL
LIN {X 0,Y 50.293,Z 607.809,A -85,B 0,C 180,E1 -29840.225,E2 -29840.225} C_VEL
LIN {X 0,Y 58.198,Z 603.923,A -85,B 0,C 180,E1 -29847.705,E2 -29847.705} C_VEL
LIN {X 0,Y 66.926,Z 598.897,A -85,B 0,C 180,E1 -29853.199,E2 -29853.199} C_VEL
LIN {X 0,Y 76.073,Z 592.565,A -85,B 0,C 180,E1 -29857.493,E2 -29857.493} C_VEL
LIN {X 0,Y 85.147,Z 584.947,A -85,B 0,C 180,E1 -29860.918,E2 -29860.918} C_VEL
LIN {X 0,Y 93.497,Z 576.578,A -85,B 0,C 180,E1 -29863.41,E2 -29863.41} C_VEL
LIN {X 0,Y 101.682,Z 566.717,A -85,B 0,C 180,E1 -29865.381,E2 -29865.381} C_VEL
LIN {X 0,Y 109.125,Z 555.599,A -85,B 0,C 180,E1 -29866.926,E2 -29866.926} C_VEL
LIN {X 0,Y 115.592,Z 543.392,A -85,B 0,C 180,E1 -29868.07,E2 -29868.07} C_VEL
LIN {X 0,Y 120.682,Z 530.584,A -85,B 0,C 180,E1 -29869.005,E2 -29869.005} C_VEL
LIN {X 0,Y 124.251,Z 517.883,A -85,B 0,C 180,E1 -29869.61,E2 -29869.61} C_VEL
LIN {X 0,Y 124.952,Z 514.628,A -85,B 0,C 180,E1 -29869.779,E2 -29869.779} C_VEL
LIN {X 0,Y 124.345,Z 511.213,A -85,B 0,C 180,E1 -29874.12,E2 -29874.12} C_VEL
LIN {X 0,Y 124.145,Z 508.937,A -85,B 0,C 180,E1 -29880,E2 -29880} C_VEL
LIN {X 0,Y 124.474,Z 511.703,A -85,B 0,C 180,E1 -29886.077,E2 -29886.077} C_VEL
LIN {X 0,Y 125.052,Z 514.643,A -85,B 0,C 180,E1 -29889.706,E2 -29889.706} C_VEL
LIN {X 0,Y 122.814,Z 524.498,A -85,B 0,C 180,E1 -29890.116,E2 -29890.116} C_VEL
LIN {X 0,Y 118.535,Z 537.47,A -85,B 0,C 180,E1 -29890.688,E2 -29890.688} C_VEL
LIN {X 0,Y 113.783,Z 548.166,A -85,B 0,C 180,E1 -29891.326,E2 -29891.326} C_VEL
LIN {X 0,Y 107.042,Z 560.069,A -85,B 0,C 180,E1 -29892.415,E2 -29892.415} C_VEL
LIN {X 0,Y 99.497,Z 570.689,A -85,B 0,C 180,E1 -29893.781,E2 -29893.781} C_VEL
LIN {X 0,Y 91.213,Z 580.266,A -85,B 0,C 180,E1 -29895.612,E2 -29895.612} C_VEL
LIN {X 0,Y 81.445,Z 589.49,A -85,B 0,C 180,E1 -29898.344,E2 -29898.344} C_VEL
LIN {X 0,Y 71.946,Z 596.915,A -85,B 0,C 180,E1 -29901.877,E2 -29901.877} C_VEL
LIN {X 0,Y 62.859,Z 602.888,A -85,B 0,C 180,E1 -29906.565,E2 -29906.565} C_VEL
LIN {X 0,Y 54.366,Z 607.616,A -85,B 0,C 180,E1 -29912.834,E2 -29912.834} C_VEL
LIN {X 0,Y 46.648,Z 611.23,A -85,B 0,C 180,E1 -29921.125,E2 -29921.125} C_VEL
LIN {X 0,Y 42.172,Z 613.096,A -85,B 0,C 180,E1 -29928.196,E2 -29928.196} C_VEL
LIN {X 0,Y 35.952,Z 615.515,A -85,B 0,C 180,E1 -29946.986,E2 -29946.986} C_VEL
LIN {X 0,Y 34.486,Z 616.137,A -85,B 0,C 180,E1 -29958.241,E2 -29958.241} C_VEL
LIN {X 0,Y 34.288,Z 616.361,A -85,B 0,C 180,E1 -29970,E2 -29970} C_VEL
LIN {X 0,Y 34.486,Z 616.117,A -85,B 0,C 180,E1 -29981.759,E2 -29981.759} C_VEL
LIN {X 0,Y 35.951,Z 615.482,A -85,B 0,C 180,E1 -29993.015,E2 -29993.015} C_VEL
LIN {X 0,Y 38.573,Z 614.457,A -85,B 0,C 180,E1 -30003.133,E2 -30003.133} C_VEL
LIN {X 0,Y 42.17,Z 613.028,A -85,B 0,C 180,E1 -30011.807,E2 -30011.807} C_VEL
LIN {X 0,Y 49.11,Z 610.057,A -85,B 0,C 180,E1 -30021.913,E2 -30021.913} C_VEL
LIN {X 0,Y 57.175,Z 606.051,A -85,B 0,C 180,E1 -30029.364,E2 -30029.364} C_VEL
LIN {X 0,Y 67.24,Z 599.994,A -85,B 0,C 180,E1 -30035.774,E2 -30035.774} C_VEL
LIN {X 0,Y 76.661,Z 593.18,A -85,B 0,C 180,E1 -30039.994,E2 -30039.994} C_VEL
LIN {X 0,Y 86.312,Z 584.872,A -85,B 0,C 180,E1 -30043.082,E2 -30043.082} C_VEL
LIN {X 0,Y 94.507,Z 576.346,A -85,B 0,C 180,E1 -30045.177,E2 -30045.177} C_VEL
LIN {X 0,Y 102.839,Z 565.824,A -85,B 0,C 180,E1 -30046.861,E2 -30046.861} C_VEL
LIN {X 0,Y 110.407,Z 553.977,A -85,B 0,C 180,E1 -30048.147,E2 -30048.147} C_VEL
LIN {X 0,Y 116.469,Z 541.673,A -85,B 0,C 180,E1 -30049.067,E2 -30049.067} C_VEL
LIN {X 0,Y 121.074,Z 529.308,A -85,B 0,C 180,E1 -30049.696,E2 -30049.696} C_VEL
LIN {X 0,Y 124.361,Z 516.801,A -85,B 0,C 180,E1 -30050.125,E2 -30050.125} C_VEL
LIN {X 0,Y 124.783,Z 514.38,A -85,B 0,C 180,E1 -30050.272,E2 -30050.272} C_VEL
LIN {X 0,Y 124.16,Z 511.105,A -85,B 0,C 180,E1 -30054.315,E2 -30054.315} C_VEL
LIN {X 0,Y 123.866,Z 508.519,A -85,B 0,C 180,E1 -30060,E2 -30060} C_VEL
LIN {X 0,Y 124.14,Z 511.404,A -85,B 0,C 180,E1 -30066.706,E2 -30066.706} C_VEL
LIN {X 0,Y 124.679,Z 514.353,A -85,B 0,C 180,E1 -30070.32,E2 -30070.32} C_VEL
LIN {X 0,Y 121.637,Z 526.54,A -85,B 0,C 180,E1 -30070.824,E2 -30070.824} C_VEL
LIN {X 0,Y 117.309,Z 538.713,A -85,B 0,C 180,E1 -30071.673,E2 -30071.673} C_VEL
LIN {X 0,Y 112.497,Z 549.03,A -85,B 0,C 180,E1 -30072.547,E2 -30072.547} C_VEL
LIN {X 0,Y 105.847,Z 560.336,A -85,B 0,C 180,E1 -30073.823,E2 -30073.823} C_VEL
LIN {X 0,Y 98.427,Z 570.522,A -85,B 0,C 180,E1 -30075.438,E2 -30075.438} C_VEL
LIN {X 0,Y 90.322,Z 579.66,A -85,B 0,C 180,E1 -30077.607,E2 -30077.607} C_VEL
LIN {X 0,Y 80.783,Z 588.541,A -85,B 0,C 180,E1 -30080.737,E2 -30080.737} C_VEL
LIN {X 0,Y 76.775,Z 591.79,A -85,B 0,C 180,E1 -30082.318,E2 -30082.318} C_VEL
LIN {X 0,Y 72.16,Z 595.056,A -85,B 0,C 180,E1 -30083.649,E2 -30083.649} C_VEL
LIN {X 0,Y 63.647,Z 599.911,A -85,B 0,C 180,E1 -30084.961,E2 -30084.961} C_VEL
LIN {X 0,Y 54.878,Z 604.112,A -85,B 0,C 180,E1 -30086.881,E2 -30086.881} C_VEL
LIN {X 0,Y 49.978,Z 606.27,A -85,B 0,C 180,E1 -30089.573,E2 -30089.573} C_VEL
LIN {X 0,Y 43.363,Z 609.021,A -85,B 0,C 180,E1 -30095.87,E2 -30095.87} C_VEL
LIN {X 0,Y 38.304,Z 610.861,A -85,B 0,C 180,E1 -30102.785,E2 -30102.785} C_VEL
LIN {X 0,Y 33.888,Z 612.24,A -85,B 0,C 180,E1 -30111.526,E2 -30111.526} C_VEL
LIN {X 0,Y 28.172,Z 613.818,A -85,B 0,C 180,E1 -30135.555,E2 -30135.555} C_VEL
LIN {X 0,Y 27.48,Z 614.037,A -85,B 0,C 180,E1 -30150,E2 -30150} C_VEL
LIN {X 0,Y 28.172,Z 613.842,A -85,B 0,C 180,E1 -30164.445,E2 -30164.445} C_VEL
LIN {X 0,Y 33.883,Z 612.294,A -85,B 0,C 180,E1 -30188.48,E2 -30188.48} C_VEL
LIN {X 0,Y 38.286,Z 610.94,A -85,B 0,C 180,E1 -30197.244,E2 -30197.244} C_VEL
LIN {X 0,Y 46.073,Z 608.076,A -85,B 0,C 180,E1 -30207.029,E2 -30207.029} C_VEL
LIN {X 0,Y 54.731,Z 604.19,A -85,B 0,C 180,E1 -30214.008,E2 -30214.008} C_VEL
LIN {X 0,Y 64.04,Z 599.163,A -85,B 0,C 180,E1 -30218.877,E2 -30218.877} C_VEL
LIN {X 0,Y 73.648,Z 592.83,A -85,B 0,C 180,E1 -30222.601,E2 -30222.601} C_VEL
LIN {X 0,Y 83.425,Z 584.92,A -85,B 0,C 180,E1 -30225.635,E2 -30225.635} C_VEL
LIN {X 0,Y 91.721,Z 576.842,A -85,B 0,C 180,E1 -30227.669,E2 -30227.669} C_VEL
LIN {X 0,Y 100.128,Z 566.98,A -85,B 0,C 180,E1 -30229.308,E2 -30229.308} C_VEL
LIN {X 0,Y 107.746,Z 555.86,A -85,B 0,C 180,E1 -30230.59,E2 -30230.59} C_VEL
LIN {X 0,Y 114.266,Z 543.803,A -85,B 0,C 180,E1 -30231.53,E2 -30231.53} C_VEL
LIN {X 0,Y 119.021,Z 532.323,A -85,B 0,C 180,E1 -30232.269,E2 -30232.269} C_VEL
LIN {X 0,Y 122.863,Z 519.364,A -85,B 0,C 180,E1 -30232.899,E2 -30232.899} C_VEL
LIN {X 0,Y 122.753,Z 517.683,A -85,B 0,C 180,E1 -30235.485,E2 -30235.485} C_VEL
LIN {X 0,Y 122.836,Z 516.071,A -85,B 0,C 180,E1 -30240,E2 -30240} C_VEL
LIN {X 0,Y 122.889,Z 518.321,A -85,B 0,C 180,E1 -30245.127,E2 -30245.127} C_VEL
LIN {X 0,Y 122.99,Z 519.402,A -85,B 0,C 180,E1 -30246.637,E2 -30246.637} C_VEL
LIN {X 0,Y 119.302,Z 532.19,A -85,B 0,C 180,E1 -30247.095,E2 -30247.095} C_VEL
LIN {X 0,Y 114.633,Z 543.742,A -85,B 0,C 180,E1 -30247.571,E2 -30247.571} C_VEL
LIN {X 0,Y 108.316,Z 555.667,A -85,B 0,C 180,E1 -30248.325,E2 -30248.325} C_VEL
LIN {X 0,Y 100.608,Z 567.165,A -85,B 0,C 180,E1 -30249.362,E2 -30249.362} C_VEL
LIN {X 0,Y 92.944,Z 576.422,A -85,B 0,C 180,E1 -30250.587,E2 -30250.587} C_VEL
LIN {X 0,Y 82.83,Z 586.365,A -85,B 0,C 180,E1 -30252.647,E2 -30252.647} C_VEL
LIN {X 0,Y 72.876,Z 594.373,A -85,B 0,C 180,E1 -30255.343,E2 -30255.343} C_VEL
LIN {X 0,Y 63.173,Z 600.796,A -85,B 0,C 180,E1 -30258.986,E2 -30258.986} C_VEL
LIN {X 0,Y 53.871,Z 605.911,A -85,B 0,C 180,E1 -30264.049,E2 -30264.049} C_VEL
LIN {X 0,Y 45.063,Z 609.885,A -85,B 0,C 180,E1 -30270.934,E2 -30270.934} C_VEL
LIN {X 0,Y 37.156,Z 612.827,A -85,B 0,C 180,E1 -30280.837,E2 -30280.837} C_VEL
LIN {X 0,Y 29.513,Z 615.247,A -85,B 0,C 180,E1 -30301.559,E2 -30301.559} C_VEL
LIN {X 0,Y 27.55,Z 615.87,A -85,B 0,C 180,E1 -30315.221,E2 -30315.221} C_VEL
LIN {X 0,Y 27.202,Z 616.095,A -85,B 0,C 180,E1 -30330,E2 -30330} C_VEL
LIN {X 0,Y 27.55,Z 615.848,A -85,B 0,C 180,E1 -30344.779,E2 -30344.779} C_VEL
LIN {X 0,Y 32.825,Z 614.188,A -85,B 0,C 180,E1 -30369.963,E2 -30369.963} C_VEL
LIN {X 0,Y 37.154,Z 612.758,A -85,B 0,C 180,E1 -30379.166,E2 -30379.166} C_VEL
LIN {X 0,Y 45.062,Z 609.788,A -85,B 0,C 180,E1 -30389.068,E2 -30389.068} C_VEL
LIN {X 0,Y 56.163,Z 604.583,A -85,B 0,C 180,E1 -30397.324,E2 -30397.324} C_VEL
LIN {X 0,Y 66.397,Z 598.606,A -85,B 0,C 180,E1 -30402.289,E2 -30402.289} C_VEL
LIN {X 0,Y 76.179,Z 591.672,A -85,B 0,C 180,E1 -30405.62,E2 -30405.62} C_VEL
LIN {X 0,Y 86.196,Z 583.001,A -85,B 0,C 180,E1 -30408.07,E2 -30408.07} C_VEL
LIN {X 0,Y 94.65,Z 574.122,A -85,B 0,C 180,E1 -30409.681,E2 -30409.681} C_VEL
LIN {X 0,Y 102.312,Z 564.376,A -85,B 0,C 180,E1 -30410.902,E2 -30410.902} C_VEL
LIN {X 0,Y 109.169,Z 553.704,A -85,B 0,C 180,E1 -30411.802,E2 -30411.802} C_VEL
LIN {X 0,Y 115.108,Z 541.924,A -85,B 0,C 180,E1 -30412.503,E2 -30412.503} C_VEL
LIN {X 0,Y 120.013,Z 529.016,A -85,B 0,C 180,E1 -30413.036,E2 -30413.036} C_VEL
LIN {X 0,Y 122.728,Z 519.125,A -85,B 0,C 180,E1 -30413.349,E2 -30413.349} C_VEL
LIN {X 0,Y 122.552,Z 517.519,A -85,B 0,C 180,E1 -30415.889,E2 -30415.889} C_VEL
LIN {X 0,Y 122.574,Z 515.69,A -85,B 0,C 180,E1 -30420,E2 -30420} C_VEL
LIN {X 0,Y 122.434,Z 516.915,A -85,B 0,C 180,E1 -30423.291,E2 -30423.291} C_VEL
LIN {X 0,Y 122.55,Z 518.495,A -85,B 0,C 180,E1 -30426.38,E2 -30426.38} C_VEL
LIN {X 0,Y 122.558,Z 519.311,A -85,B 0,C 180,E1 -30427.253,E2 -30427.253} C_VEL
LIN {X 0,Y 119.488,Z 529.945,A -85,B 0,C 180,E1 -30427.69,E2 -30427.69} C_VEL
LIN {X 0,Y 114.754,Z 542.068,A -85,B 0,C 180,E1 -30428.422,E2 -30428.422} C_VEL
LIN {X 0,Y 108.629,Z 553.862,A -85,B 0,C 180,E1 -30429.388,E2 -30429.388} C_VEL
LIN {X 0,Y 101.007,Z 565.393,A -85,B 0,C 180,E1 -30430.645,E2 -30430.645} C_VEL
LIN {X 0,Y 93.425,Z 574.683,A -85,B 0,C 180,E1 -30432.064,E2 -30432.064} C_VEL
LIN {X 0,Y 85.122,Z 583.135,A -85,B 0,C 180,E1 -30434.052,E2 -30434.052} C_VEL
LIN {X 0,Y 75.305,Z 591.354,A -85,B 0,C 180,E1 -30436.947,E2 -30436.947} C_VEL
LIN {X 0,Y 67.26,Z 596.976,A -85,B 0,C 180,E1 -30439.884,E2 -30439.884} C_VEL
LIN {X 0,Y 57.821,Z 602.459,A -85,B 0,C 180,E1 -30444.274,E2 -30444.274} C_VEL
LIN {X 0,Y 49.978,Z 606.27,A -85,B 0,C 180,E1 -30449.573,E2 -30449.573} C_VEL
LIN {X 0,Y 45.133,Z 608.23,A -85,B 0,C 180,E1 -30452.907,E2 -30452.907} C_VEL
LIN {X 0,Y 36.339,Z 610.943,A -85,B 0,C 180,E1 -30458.143,E2 -30458.143} C_VEL
LIN {X 0,Y 29.405,Z 612.546,A -85,B 0,C 180,E1 -30464.402,E2 -30464.402} C_VEL
LIN {X 0,Y 25.015,Z 613.368,A -85,B 0,C 180,E1 -30472.647,E2 -30472.647} C_VEL
LIN {X 0,Y 23.888,Z 613.559,A -85,B 0,C 180,E1 -30476.425,E2 -30476.425} C_VEL
LIN {X 0,Y 20.384,Z 614.304,A -85,B 0,C 180,E1 -30510,E2 -30510} C_VEL
LIN {X 0,Y 21.388,Z 614.108,A -85,B 0,C 180,E1 -30529.183,E2 -30529.183} C_VEL
LIN {X 0,Y 28.662,Z 612.561,A -85,B 0,C 180,E1 -30557.358,E2 -30557.358} C_VEL
LIN {X 0,Y 33.877,Z 611.206,A -85,B 0,C 180,E1 -30566.078,E2 -30566.078} C_VEL
LIN {X 0,Y 42.628,Z 608.342,A -85,B 0,C 180,E1 -30575.062,E2 -30575.062} C_VEL
LIN {X 0,Y 52.012,Z 604.456,A -85,B 0,C 180,E1 -30581.057,E2 -30581.057} C_VEL
LIN {X 0,Y 61.838,Z 599.429,A -85,B 0,C 180,E1 -30585.02,E2 -30585.02} C_VEL
LIN {X 0,Y 71.845,Z 593.095,A -85,B 0,C 180,E1 -30588.014,E2 -30588.014} C_VEL
LIN {X 0,Y 81.954,Z 585.182,A -85,B 0,C 180,E1 -30590.457,E2 -30590.457} C_VEL
LIN {X 0,Y 90.473,Z 577.106,A -85,B 0,C 180,E1 -30592.056,E2 -30592.056} C_VEL
LIN {X 0,Y 99.059,Z 567.244,A -85,B 0,C 180,E1 -30593.338,E2 -30593.338} C_VEL
LIN {X 0,Y 106.815,Z 556.123,A -85,B 0,C 180,E1 -30594.348,E2 -30594.348} C_VEL
LIN {X 0,Y 112.869,Z 545.218,A -85,B 0,C 180,E1 -30595.034,E2 -30595.034} C_VEL
LIN {X 0,Y 117.951,Z 533.432,A -85,B 0,C 180,E1 -30595.633,E2 -30595.633} C_VEL
LIN {X 0,Y 120.902,Z 524.435,A -85,B 0,C 180,E1 -30596.012,E2 -30596.012} C_VEL
LIN {X 0,Y 121.08,Z 523.11,A -85,B 0,C 180,E1 -30600,E2 -30600} C_VEL
LIN {X 0,Y 120.994,Z 524.428,A -85,B 0,C 180,E1 -30603.444,E2 -30603.444} C_VEL
LIN {X 0,Y 116.639,Z 537.21,A -85,B 0,C 180,E1 -30603.837,E2 -30603.837} C_VEL
LIN {X 0,Y 110.994,Z 549.296,A -85,B 0,C 180,E1 -30604.25,E2 -30604.25} C_VEL
LIN {X 0,Y 104.041,Z 560.837,A -85,B 0,C 180,E1 -30604.904,E2 -30604.904} C_VEL
LIN {X 0,Y 96.233,Z 571.234,A -85,B 0,C 180,E1 -30605.716,E2 -30605.716} C_VEL
LIN {X 0,Y 88.45,Z 579.736,A -85,B 0,C 180,E1 -30606.689,E2 -30606.689} C_VEL
LIN {X 0,Y 78.138,Z 588.957,A -85,B 0,C 180,E1 -30608.367,E2 -30608.367} C_VEL
LIN {X 0,Y 67.932,Z 596.382,A -85,B 0,C 180,E1 -30610.637,E2 -30610.637} C_VEL
LIN {X 0,Y 57.898,Z 602.354,A -85,B 0,C 180,E1 -30613.815,E2 -30613.815} C_VEL
LIN {X 0,Y 48.153,Z 607.082,A -85,B 0,C 180,E1 -30618.439,E2 -30618.439} C_VEL
LIN {X 0,Y 38.789,Z 610.696,A -85,B 0,C 180,E1 -30625.053,E2 -30625.053} C_VEL
LIN {X 0,Y 32.937,Z 612.56,A -85,B 0,C 180,E1 -30631.406,E2 -30631.406} C_VEL
LIN {X 0,Y 23.49,Z 614.979,A -85,B 0,C 180,E1 -30653.248,E2 -30653.248} C_VEL
LIN {X 0,Y 20.753,Z 615.602,A -85,B 0,C 180,E1 -30670.206,E2 -30670.206} C_VEL
LIN {X 0,Y 20.084,Z 615.827,A -85,B 0,C 180,E1 -30690,E2 -30690} C_VEL
LIN {X 0,Y 20.752,Z 615.581,A -85,B 0,C 180,E1 -30709.795,E2 -30709.795} C_VEL
LIN {X 0,Y 27.739,Z 613.919,A -85,B 0,C 180,E1 -30739.47,E2 -30739.47} C_VEL
LIN {X 0,Y 32.935,Z 612.489,A -85,B 0,C 180,E1 -30748.598,E2 -30748.598} C_VEL
LIN {X 0,Y 41.847,Z 609.519,A -85,B 0,C 180,E1 -30757.469,E2 -30757.469} C_VEL
LIN {X 0,Y 51.386,Z 605.511,A -85,B 0,C 180,E1 -30763.208,E2 -30763.208} C_VEL
LIN {X 0,Y 62.914,Z 599.352,A -85,B 0,C 180,E1 -30767.801,E2 -30767.801} C_VEL
LIN {X 0,Y 73.028,Z 592.641,A -85,B 0,C 180,E1 -30770.544,E2 -30770.544} C_VEL
LIN {X 0,Y 83.294,Z 584.332,A -85,B 0,C 180,E1 -30772.478,E2 -30772.478} C_VEL
LIN {X 0,Y 91.905,Z 575.806,A -85,B 0,C 180,E1 -30773.768,E2 -30773.768} C_VEL
LIN {X 0,Y 100.564,Z 565.281,A -85,B 0,C 180,E1 -30774.779,E2 -30774.779} C_VEL
LIN {X 0,Y 108.383,Z 553.432,A -85,B 0,C 180,E1 -30775.525,E2 -30775.525} C_VEL
